LIN {X 0,Y 361.951,Z 263.021,A -85,B 0,C 180,E1 -13113.474,E2 -13113.474} C_VEL
LIN {X 0,Y 361.885,Z 263.028,A -85,B 0,C 180,E1 -13117.143,E2 -13117.143} C_VEL
LIN {X 0,Y 361.906,Z 263.025,A -85,B 0,C 180,E1 -13120.722,E2 -13120.722} C_VEL
LIN {X 0,Y 361.927,Z 263.025,A -85,B 0,C 180,E1 -13123.064,E2 -13123.064} C_VEL
LIN {X 0,Y 361.993,Z 263.017,A -85,B 0,C 180,E1 -13126.526,E2 -13126.526} C_VEL
LIN {X 0,Y 362.025,Z 263.015,A -85,B 0,C 180,E1 -13129.936,E2 -13129.936} C_VEL
LIN {X 0,Y 362.155,Z 262.991,A -85,B 0,C 180,E1 -13133.312,E2 -13133.312} C_VEL
LIN {X 0,Y 362.275,Z 262.98,A -85,B 0,C 180,E1 -13137.775,E2 -13137.775} C_VEL
LIN {X 0,Y 362.421,Z 262.962,A -85,B 0,C 180,E1 -13139.999,E2 -13139.999} C_VEL
LIN {X 0,Y 362.274,Z 262.978,A -85,B 0,C 180,E1 -13142.222,E2 -13142.222} C_VEL
LIN {X 0,Y 362.153,Z 262.994,A -85,B 0,C 180,E1 -13146.685,E2 -13146.685} C_VEL
LIN {X 0,Y 362.021,Z 263.007,A -85,B 0,C 180,E1 -13150.061,E2 -13150.061} C_VEL
LIN {X 0,Y 361.987,Z 263.012,A -85,B 0,C 180,E1 -13153.897,E2 -13153.897} C_VEL
LIN {X 0,Y 361.957,Z 263.018,A -85,B 0,C 180,E1 -13157.938,E2 -13157.938} C_VEL
LIN {X 0,Y 361.891,Z 263.03,A -85,B 0,C 180,E1 -13161.651,E2 -13161.651} C_VEL
LIN {X 0,Y 361.917,Z 263.028,A -85,B 0,C 180,E1 -13165.289,E2 -13165.289} C_VEL
LIN {X 0,Y 361.91,Z 263.028,A -85,B 0,C 180,E1 -13167.777,E2 -13167.777} C_VEL
LIN {X 0,Y 361.834,Z 263.024,A -85,B 0,C 180,E1 -13171.284,E2 -13171.284} C_VEL
LIN {X 0,Y 361.841,Z 263.03,A -85,B 0,C 180,E1 -13174.279,E2 -13174.279} C_VEL
LIN {X 0,Y 361.859,Z 263.037,A -85,B 0,C 180,E1 -13177.224,E2 -13177.224} C_VEL
LIN {X 0,Y 361.892,Z 263.034,A -85,B 0,C 180,E1 -13180.767,E2 -13180.767} C_VEL
LIN {X 0,Y 361.948,Z 263.04,A -85,B 0,C 180,E1 -13184.914,E2 -13184.914} C_VEL
LIN {X 0,Y 364.418,Z 272.898,A -85,B 0,C 180,E1 -13187.831,E2 -13187.831} C_VEL
LIN {X 0,Y 372.996,Z 290.807,A -85,B 0,C 180,E1 -13189.061,E2 -13189.061} C_VEL
LIN {X 0,Y 377.155,Z 300.817,A -85,B 0,C 180,E1 -13189.66,E2 -13189.66} C_VEL
LIN {X 0,Y 377.876,Z 305.295,A -85,B 0,C 180,E1 -13189.822,E2 -13189.822} C_VEL
LIN {X 0,Y 375.211,Z 409.637,A -85,B 0,C 180,E1 -13191.888,E2 -13191.888} C_VEL
LIN {X 0,Y 374.417,Z 423.861,A -85,B 0,C 180,E1 -13192.384,E2 -13192.384} C_VEL
LIN {X 0,Y 373.309,Z 436.994,A -85,B 0,C 180,E1 -13193.041,E2 -13193.041} C_VEL
LIN {X 0,Y 372.043,Z 450.844,A -85,B 0,C 180,E1 -13193.989,E2 -13193.989} C_VEL
LIN {X 0,Y 370.563,Z 463.295,A -85,B 0,C 180,E1 -13195.075,E2 -13195.075} C_VEL
LIN {X 0,Y 369.18,Z 473.466,A -85,B 0,C 180,E1 -13196.165,E2 -13196.165} C_VEL
LIN {X 0,Y 367.475,Z 484.71,A -85,B 0,C 180,E1 -13197.623,E2 -13197.623} C_VEL
LIN {X 0,Y 366.018,Z 494.031,A -85,B 0,C 180,E1 -13199.095,E2 -13199.095} C_VEL
LIN {X 0,Y 364.568,Z 503.314,A -85,B 0,C 180,E1 -13200.873,E2 -13200.873} C_VEL
LIN {X 0,Y 363.209,Z 511.817,A -85,B 0,C 180,E1 -13202.88,E2 -13202.88} C_VEL
LIN {X 0,Y 362.229,Z 518.114,A -85,B 0,C 180,E1 -13204.733,E2 -13204.733} C_VEL
LIN {X 0,Y 361.511,Z 523.028,A -85,B 0,C 180,E1 -13206.533,E2 -13206.533} C_VEL
LIN {X 0,Y 360.993,Z 526.84,A -85,B 0,C 180,E1 -13208.291,E2 -13208.291} C_VEL
LIN {X 0,Y 360.753,Z 528.882,A -85,B 0,C 180,E1 -13209.473,E2 -13209.473} C_VEL
LIN {X 0,Y 360.334,Z 531.796,A -85,B 0,C 180,E1 -13211.817,E2 -13211.817} C_VEL
LIN {X 0,Y 360.169,Z 533.243,A -85,B 0,C 180,E1 -13214.147,E2 -13214.147} C_VEL
LIN {X 0,Y 360.14,Z 533.273,A -85,B 0,C 180,E1 -13216.457,E2 -13216.457} C_VEL
LIN {X 0,Y 360.223,Z 532.756,A -85,B 0,C 180,E1 -13217.608,E2 -13217.608} C_VEL
LIN {X 0,Y 360.232,Z 530.689,A -85,B 0,C 180,E1 -13219.888,E2 -13219.888} C_VEL
LIN {X 0,Y 360.554,Z 527.2,A -85,B 0,C 180,E1 -13222.158,E2 -13222.158} C_VEL
LIN {X 0,Y 360.956,Z 522.221,A -85,B 0,C 180,E1 -13224.414,E2 -13224.414} C_VEL
LIN {X 0,Y 361.337,Z 517.421,A -85,B 0,C 180,E1 -13226.097,E2 -13226.097} C_VEL
LIN {X 0,Y 361.974,Z 510.498,A -85,B 0,C 180,E1 -13228.053,E2 -13228.053} C_VEL
LIN {X 0,Y 362.819,Z 503.263,A -85,B 0,C 180,E1 -13229.723,E2 -13229.723} C_VEL
LIN {X 0,Y 363.876,Z 494.569,A -85,B 0,C 180,E1 -13231.384,E2 -13231.384} C_VEL
LIN {X 0,Y 365.098,Z 484.058,A -85,B 0,C 180,E1 -13233.035,E2 -13233.035} C_VEL
LIN {X 0,Y 366.459,Z 472.289,A -85,B 0,C 180,E1 -13234.537,E2 -13234.537} C_VEL
LIN {X 0,Y 367.69,Z 460.24,A -85,B 0,C 180,E1 -13235.784,E2 -13235.784} C_VEL
LIN {X 0,Y 368.854,Z 447.486,A -85,B 0,C 180,E1 -13236.839,E2 -13236.839} C_VEL
LIN {X 0,Y 369.768,Z 433.835,A -85,B 0,C 180,E1 -13237.714,E2 -13237.714} C_VEL
LIN {X 0,Y 370.561,Z 419.368,A -85,B 0,C 180,E1 -13238.384,E2 -13238.384} C_VEL
LIN {X 0,Y 371.08,Z 405.045,A -85,B 0,C 180,E1 -13238.818,E2 -13238.818} C_VEL
LIN {X 0,Y 371.751,Z 371.974,A -85,B 0,C 180,E1 -13239.465,E2 -13239.465} C_VEL
LIN {X 0,Y 371.242,Z 366.164,A -85,B 0,C 180,E1 -13239.612,E2 -13239.612} C_VEL
LIN {X 0,Y 366.276,Z 347.449,A -85,B 0,C 180,E1 -13240.285,E2 -13240.285} C_VEL
LIN {X 0,Y 365.76,Z 341.639,A -85,B 0,C 180,E1 -13240.437,E2 -13240.437} C_VEL
LIN {X 0,Y 366.376,Z 302.629,A -85,B 0,C 180,E1 -13241.213,E2 -13241.213} C_VEL
LIN {X 0,Y 363.787,Z 291.177,A -85,B 0,C 180,E1 -13241.617,E2 -13241.617} C_VEL
LIN {X 0,Y 356.731,Z 272.196,A -85,B 0,C 180,E1 -13242.516,E2 -13242.516} C_VEL
LIN {X 0,Y 354.914,Z 263.908,A -85,B 0,C 180,E1 -13244.744,E2 -13244.744} C_VEL
LIN {X 0,Y 354.895,Z 263.9,A -85,B 0,C 180,E1 -13248.472,E2 -13248.472} C_VEL
LIN {X 0,Y 354.826,Z 263.911,A -85,B 0,C 180,E1 -13252.106,E2 -13252.106} C_VEL
LIN {X 0,Y 354.886,Z 263.905,A -85,B 0,C 180,E1 -13255.828,E2 -13255.828} C_VEL
LIN {X 0,Y 354.842,Z 263.911,A -85,B 0,C 180,E1 -13259.679,E2 -13259.679} C_VEL
LIN {X 0,Y 354.793,Z 263.916,A -85,B 0,C 180,E1 -13263.703,E2 -13263.703} C_VEL
LIN {X 0,Y 354.789,Z 263.912,A -85,B 0,C 180,E1 -13266.46,E2 -13266.46} C_VEL
LIN {X 0,Y 354.812,Z 263.916,A -85,B 0,C 180,E1 -13269.424,E2 -13269.424} C_VEL
LIN {X 0,Y 354.83,Z 263.909,A -85,B 0,C 180,E1 -13272.877,E2 -13272.877} C_VEL
LIN {X 0,Y 354.853,Z 263.904,A -85,B 0,C 180,E1 -13276.12,E2 -13276.12} C_VEL
LIN {X 0,Y 354.844,Z 263.911,A -85,B 0,C 180,E1 -13279.19,E2 -13279.19} C_VEL
LIN {X 0,Y 354.797,Z 263.912,A -85,B 0,C 180,E1 -13282.403,E2 -13282.403} C_VEL
LIN {X 0,Y 354.801,Z 263.914,A -85,B 0,C 180,E1 -13284.942,E2 -13284.942} C_VEL
LIN {X 0,Y 354.782,Z 263.914,A -85,B 0,C 180,E1 -13288.406,E2 -13288.406} C_VEL
LIN {X 0,Y 354.843,Z 263.906,A -85,B 0,C 180,E1 -13291.621,E2 -13291.621} C_VEL
LIN {X 0,Y 354.889,Z 263.9,A -85,B 0,C 180,E1 -13294.174,E2 -13294.174} C_VEL
LIN {X 0,Y 354.824,Z 263.908,A -85,B 0,C 180,E1 -13297.895,E2 -13297.895} C_VEL
LIN {X 0,Y 354.913,Z 263.897,A -85,B 0,C 180,E1 -13301.893,E2 -13301.893} C_VEL
LIN {X 0,Y 354.934,Z 263.895,A -85,B 0,C 180,E1 -13305.983,E2 -13305.983} C_VEL
LIN {X 0,Y 354.97,Z 263.89,A -85,B 0,C 180,E1 -13309.737,E2 -13309.737} C_VEL
LIN {X 0,Y 355.119,Z 263.872,A -85,B 0,C 180,E1 -13313.182,E2 -13313.182} C_VEL
LIN {X 0,Y 355.239,Z 263.857,A -85,B 0,C 180,E1 -13317.734,E2 -13317.734} C_VEL
LIN {X 0,Y 355.39,Z 263.839,A -85,B 0,C 180,E1 -13320.002,E2 -13320.002} C_VEL
LIN {X 0,Y 355.239,Z 263.86,A -85,B 0,C 180,E1 -13322.269,E2 -13322.269} C_VEL
LIN {X 0,Y 355.12,Z 263.873,A -85,B 0,C 180,E1 -13326.821,E2 -13326.821} C_VEL
LIN {X 0,Y 354.973,Z 263.896,A -85,B 0,C 180,E1 -13330.266,E2 -13330.266} C_VEL
LIN {X 0,Y 354.939,Z 263.897,A -85,B 0,C 180,E1 -13334.02,E2 -13334.02} C_VEL
LIN {X 0,Y 354.919,Z 263.902,A -85,B 0,C 180,E1 -13338.11,E2 -13338.11} C_VEL
LIN {X 0,Y 354.814,Z 263.915,A -85,B 0,C 180,E1 -13342.109,E2 -13342.109} C_VEL
LIN {X 0,Y 354.896,Z 263.903,A -85,B 0,C 180,E1 -13345.829,E2 -13345.829} C_VEL
LIN {X 0,Y 354.853,Z 263.908,A -85,B 0,C 180,E1 -13349.68,E2 -13349.68} C_VEL
LIN {X 0,Y 354.83,Z 263.912,A -85,B 0,C 180,E1 -13353.684,E2 -13353.684} C_VEL
LIN {X 0,Y 354.798,Z 263.912,A -85,B 0,C 180,E1 -13356.461,E2 -13356.461} C_VEL
LIN {X 0,Y 354.824,Z 263.911,A -85,B 0,C 180,E1 -13359.425,E2 -13359.425} C_VEL
LIN {X 0,Y 354.788,Z 263.913,A -85,B 0,C 180,E1 -13362.868,E2 -13362.868} C_VEL
LIN {X 0,Y 354.768,Z 263.917,A -85,B 0,C 180,E1 -13366.105,E2 -13366.105} C_VEL
LIN {X 0,Y 354.788,Z 263.915,A -85,B 0,C 180,E1 -13369.18,E2 -13369.18} C_VEL
LIN {X 0,Y 354.808,Z 263.91,A -85,B 0,C 180,E1 -13372.404,E2 -13372.404} C_VEL
LIN {X 0,Y 354.814,Z 263.911,A -85,B 0,C 180,E1 -13374.942,E2 -13374.942} C_VEL
LIN {X 0,Y 354.846,Z 264.002,A -85,B 0,C 180,E1 -13377.589,E2 -13377.589} C_VEL
LIN {X 0,Y 357.921,Z 277.781,A -85,B 0,C 180,E1 -13380.924,E2 -13380.924} C_VEL
LIN {X 0,Y 359.764,Z 286.653,A -85,B 0,C 180,E1 -13382.988,E2 -13382.988} C_VEL
LIN {X 0,Y 359.785,Z 290.384,A -85,B 0,C 180,E1 -13383.74,E2 -13383.74} C_VEL
LIN {X 0,Y 366.128,Z 328.545,A -85,B 0,C 180,E1 -13384.945,E2 -13384.945} C_VEL
LIN {X 0,Y 364.125,Z 427.883,A -85,B 0,C 180,E1 -13386.918,E2 -13386.918} C_VEL
LIN {X 0,Y 363.381,Z 442.676,A -85,B 0,C 180,E1 -13387.432,E2 -13387.432} C_VEL
LIN {X 0,Y 362.317,Z 456.75,A -85,B 0,C 180,E1 -13388.15,E2 -13388.15} C_VEL
LIN {X 0,Y 361.201,Z 470.732,A -85,B 0,C 180,E1 -13389.125,E2 -13389.125} C_VEL
LIN {X 0,Y 359.782,Z 483.977,A -85,B 0,C 180,E1 -13390.308,E2 -13390.308} C_VEL
LIN {X 0,Y 358.365,Z 496.401,A -85,B 0,C 180,E1 -13391.713,E2 -13391.713} C_VEL
LIN {X 0,Y 357.116,Z 506.619,A -85,B 0,C 180,E1 -13393.126,E2 -13393.126} C_VEL
LIN {X 0,Y 355.983,Z 516.769,A -85,B 0,C 180,E1 -13394.836,E2 -13394.836} C_VEL
LIN {X 0,Y 355.17,Z 525.186,A -85,B 0,C 180,E1 -13396.556,E2 -13396.556} C_VEL
LIN {X 0,Y 354.276,Z 533.205,A -85,B 0,C 180,E1 -13398.558,E2 -13398.558} C_VEL
LIN {X 0,Y 353.783,Z 538.828,A -85,B 0,C 180,E1 -13400.279,E2 -13400.279} C_VEL
LIN {X 0,Y 353.417,Z 544.71,A -85,B 0,C 180,E1 -13402.573,E2 -13402.573} C_VEL
LIN {X 0,Y 353.265,Z 548.085,A -85,B 0,C 180,E1 -13404.291,E2 -13404.291} C_VEL
LIN {X 0,Y 353.207,Z 551.233,A -85,B 0,C 180,E1 -13406.578,E2 -13406.578} C_VEL
LIN {X 0,Y 353.221,Z 552.988,A -85,B 0,C 180,E1 -13408.86,E2 -13408.86} C_VEL
LIN {X 0,Y 353.263,Z 553.359,A -85,B 0,C 180,E1 -13410,E2 -13410} C_VEL
LIN {X 0,Y 353.167,Z 553.092,A -85,B 0,C 180,E1 -13412.281,E2 -13412.281} C_VEL
LIN {X 0,Y 353.242,Z 551.497,A -85,B 0,C 180,E1 -13414.564,E2 -13414.564} C_VEL
LIN {X 0,Y 353.396,Z 548.542,A -85,B 0,C 180,E1 -13416.853,E2 -13416.853} C_VEL
LIN {X 0,Y 353.775,Z 544.152,A -85,B 0,C 180,E1 -13419.144,E2 -13419.144} C_VEL
LIN {X 0,Y 354.421,Z 538.215,A -85,B 0,C 180,E1 -13421.437,E2 -13421.437} C_VEL
LIN {X 0,Y 355.514,Z 531.558,A -85,B 0,C 180,E1 -13423.431,E2 -13423.431} C_VEL
LIN {X 0,Y 356.675,Z 523.31,A -85,B 0,C 180,E1 -13425.426,E2 -13425.426} C_VEL
LIN {X 0,Y 358.084,Z 514.738,A -85,B 0,C 180,E1 -13427.121,E2 -13427.121} C_VEL
LIN {X 0,Y 359.812,Z 504.379,A -85,B 0,C 180,E1 -13428.801,E2 -13428.801} C_VEL
LIN {X 0,Y 361.661,Z 492.828,A -85,B 0,C 180,E1 -13430.325,E2 -13430.325} C_VEL
LIN {X 0,Y 363.336,Z 481.321,A -85,B 0,C 180,E1 -13431.562,E2 -13431.562} C_VEL
LIN {X 0,Y 364.933,Z 468.715,A -85,B 0,C 180,E1 -13432.653,E2 -13432.653} C_VEL
LIN {X 0,Y 366.396,Z 455.701,A -85,B 0,C 180,E1 -13433.528,E2 -13433.528} C_VEL
LIN {X 0,Y 367.728,Z 441.697,A -85,B 0,C 180,E1 -13434.224,E2 -13434.224} C_VEL
LIN {X 0,Y 368.599,Z 428.135,A -85,B 0,C 180,E1 -13434.688,E2 -13434.688} C_VEL
LIN {X 0,Y 371.103,Z 329.531,A -85,B 0,C 180,E1 -13436.683,E2 -13436.683} C_VEL
LIN {X 0,Y 366.385,Z 305.41,A -85,B 0,C 180,E1 -13437.663,E2 -13437.663} C_VEL
LIN {X 0,Y 364.205,Z 296.489,A -85,B 0,C 180,E1 -13438.077,E2 -13438.077} C_VEL
LIN {X 0,Y 361.196,Z 289.435,A -85,B 0,C 180,E1 -13438.551,E2 -13438.551} C_VEL
LIN {X 0,Y 358.485,Z 277.757,A -85,B 0,C 180,E1 -13441.628,E2 -13441.628} C_VEL
LIN {X 0,Y 355.393,Z 265.851,A -85,B 0,C 180,E1 -13444.992,E2 -13444.992} C_VEL
LIN {X 0,Y 354.837,Z 263.916,A -85,B 0,C 180,E1 -13445.601,E2 -13445.601} C_VEL
LIN {X 0,Y 354.825,Z 263.917,A -85,B 0,C 180,E1 -13449.422,E2 -13449.422} C_VEL
LIN {X 0,Y 354.834,Z 263.912,A -85,B 0,C 180,E1 -13452.874,E2 -13452.874} C_VEL
LIN {X 0,Y 354.783,Z 263.916,A -85,B 0,C 180,E1 -13456.105,E2 -13456.105} C_VEL
LIN {X 0,Y 354.786,Z 263.916,A -85,B 0,C 180,E1 -13459.177,E2 -13459.177} C_VEL
LIN {X 0,Y 354.805,Z 263.909,A -85,B 0,C 180,E1 -13462.401,E2 -13462.401} C_VEL
LIN {X 0,Y 354.809,Z 263.893,A -85,B 0,C 180,E1 -13464.939,E2 -13464.939} C_VEL
LIN {X 0,Y 354.79,Z 263.909,A -85,B 0,C 180,E1 -13468.404,E2 -13468.404} C_VEL
LIN {X 0,Y 354.85,Z 263.906,A -85,B 0,C 180,E1 -13471.618,E2 -13471.618} C_VEL
LIN {X 0,Y 354.895,Z 263.903,A -85,B 0,C 180,E1 -13474.171,E2 -13474.171} C_VEL
LIN {X 0,Y 354.83,Z 263.913,A -85,B 0,C 180,E1 -13477.892,E2 -13477.892} C_VEL
LIN {X 0,Y 354.918,Z 263.901,A -85,B 0,C 180,E1 -13481.89,E2 -13481.89} C_VEL
LIN {X 0,Y 354.937,Z 263.898,A -85,B 0,C 180,E1 -13485.98,E2 -13485.98} C_VEL
LIN {X 0,Y 354.971,Z 263.894,A -85,B 0,C 180,E1 -13489.734,E2 -13489.734} C_VEL
LIN {X 0,Y 355.119,Z 263.866,A -85,B 0,C 180,E1 -13493.179,E2 -13493.179} C_VEL
LIN {X 0,Y 355.238,Z 263.855,A -85,B 0,C 180,E1 -13497.731,E2 -13497.731} C_VEL
LIN {X 0,Y 355.391,Z 263.838,A -85,B 0,C 180,E1 -13499.998,E2 -13499.998} C_VEL
LIN {X 0,Y 355.237,Z 263.855,A -85,B 0,C 180,E1 -13502.266,E2 -13502.266} C_VEL
LIN {X 0,Y 355.117,Z 263.871,A -85,B 0,C 180,E1 -13506.818,E2 -13506.818} C_VEL
LIN {X 0,Y 354.968,Z 263.886,A -85,B 0,C 180,E1 -13510.263,E2 -13510.263} C_VEL
LIN {X 0,Y 354.932,Z 263.891,A -85,B 0,C 180,E1 -13514.017,E2 -13514.017} C_VEL
LIN {X 0,Y 354.913,Z 263.896,A -85,B 0,C 180,E1 -13518.108,E2 -13518.108} C_VEL
LIN {X 0,Y 354.833,Z 263.909,A -85,B 0,C 180,E1 -13522.104,E2 -13522.104} C_VEL
LIN {X 0,Y 354.888,Z 263.903,A -85,B 0,C 180,E1 -13525.826,E2 -13525.826} C_VEL
LIN {X 0,Y 354.842,Z 263.901,A -85,B 0,C 180,E1 -13529.677,E2 -13529.677} C_VEL
LIN {X 0,Y 354.793,Z 263.915,A -85,B 0,C 180,E1 -13533.701,E2 -13533.701} C_VEL
LIN {X 0,Y 354.788,Z 263.912,A -85,B 0,C 180,E1 -13536.458,E2 -13536.458} C_VEL
LIN {X 0,Y 354.811,Z 263.905,A -85,B 0,C 180,E1 -13539.423,E2 -13539.423} C_VEL
LIN {X 0,Y 354.828,Z 263.907,A -85,B 0,C 180,E1 -13542.876,E2 -13542.876} C_VEL
LIN {X 0,Y 354.919,Z 264.059,A -85,B 0,C 180,E1 -13544.327,E2 -13544.327} C_VEL
LIN {X 0,Y 357.304,Z 273.246,A -85,B 0,C 180,E1 -13547.109,E2 -13547.109} C_VEL
LIN {X 0,Y 366.119,Z 291.157,A -85,B 0,C 180,E1 -13548.418,E2 -13548.418} C_VEL
LIN {X 0,Y 371.246,Z 303.218,A -85,B 0,C 180,E1 -13549.176,E2 -13549.176} C_VEL
LIN {X 0,Y 371.747,Z 306.001,A -85,B 0,C 180,E1 -13549.284,E2 -13549.284} C_VEL
LIN {X 0,Y 368.982,Z 409.593,A -85,B 0,C 180,E1 -13551.367,E2 -13551.367} C_VEL
LIN {X 0,Y 368.105,Z 424.319,A -85,B 0,C 180,E1 -13551.888,E2 -13551.888} C_VEL
LIN {X 0,Y 366.87,Z 438.537,A -85,B 0,C 180,E1 -13552.626,E2 -13552.626} C_VEL
LIN {X 0,Y 365.619,Z 451.321,A -85,B 0,C 180,E1 -13553.528,E2 -13553.528} C_VEL
LIN {X 0,Y 364.088,Z 463.555,A -85,B 0,C 180,E1 -13554.614,E2 -13554.614} C_VEL
LIN {X 0,Y 362.552,Z 474.341,A -85,B 0,C 180,E1 -13555.796,E2 -13555.796} C_VEL
LIN {X 0,Y 360.778,Z 485.47,A -85,B 0,C 180,E1 -13557.278,E2 -13557.278} C_VEL
LIN {X 0,Y 359.246,Z 494.693,A -85,B 0,C 180,E1 -13558.774,E2 -13558.774} C_VEL
LIN {X 0,Y 357.716,Z 503.898,A -85,B 0,C 180,E1 -13560.583,E2 -13560.583} C_VEL
LIN {X 0,Y 356.333,Z 512.078,A -85,B 0,C 180,E1 -13562.561,E2 -13562.561} C_VEL
LIN {X 0,Y 355.403,Z 517.622,A -85,B 0,C 180,E1 -13564.213,E2 -13564.213} C_VEL
LIN {X 0,Y 354.57,Z 522.958,A -85,B 0,C 180,E1 -13566.16,E2 -13566.16} C_VEL
LIN {X 0,Y 353.878,Z 527.737,A -85,B 0,C 180,E1 -13568.445,E2 -13568.445} C_VEL
LIN {X 0,Y 353.491,Z 530.451,A -85,B 0,C 180,E1 -13570.246,E2 -13570.246} C_VEL
LIN {X 0,Y 353.179,Z 532.748,A -85,B 0,C 180,E1 -13572.634,E2 -13572.634} C_VEL
LIN {X 0,Y 353.04,Z 533.608,A -85,B 0,C 180,E1 -13575.002,E2 -13575.002} C_VEL
LIN {X 0,Y 353.124,Z 533.069,A -85,B 0,C 180,E1 -13577.354,E2 -13577.354} C_VEL
LIN {X 0,Y 353.129,Z 531.156,A -85,B 0,C 180,E1 -13579.682,E2 -13579.682} C_VEL
LIN {X 0,Y 353.44,Z 527.799,A -85,B 0,C 180,E1 -13581.999,E2 -13581.999} C_VEL
LIN {X 0,Y 353.675,Z 524.86,A -85,B 0,C 180,E1 -13583.478,E2 -13583.478} C_VEL
LIN {X 0,Y 354.03,Z 519.936,A -85,B 0,C 180,E1 -13585.446,E2 -13585.446} C_VEL
LIN {X 0,Y 354.657,Z 513.585,A -85,B 0,C 180,E1 -13587.445,E2 -13587.445} C_VEL
LIN {X 0,Y 355.611,Z 505.686,A -85,B 0,C 180,E1 -13589.434,E2 -13589.434} C_VEL
LIN {X 0,Y 356.592,Z 497.444,A -85,B 0,C 180,E1 -13591.129,E2 -13591.129} C_VEL
LIN {X 0,Y 357.806,Z 487.525,A -85,B 0,C 180,E1 -13592.815,E2 -13592.815} C_VEL
LIN {X 0,Y 359.162,Z 476.493,A -85,B 0,C 180,E1 -13594.349,E2 -13594.349} C_VEL
LIN {X 0,Y 360.387,Z 465.534,A -85,B 0,C 180,E1 -13595.596,E2 -13595.596} C_VEL
LIN {X 0,Y 361.491,Z 453.705,A -85,B 0,C 180,E1 -13596.699,E2 -13596.699} C_VEL
LIN {X 0,Y 362.593,Z 440.692,A -85,B 0,C 180,E1 -13597.658,E2 -13597.658} C_VEL
LIN {X 0,Y 363.51,Z 426.527,A -85,B 0,C 180,E1 -13598.442,E2 -13598.442} C_VEL
LIN {X 0,Y 364.127,Z 412.525,A -85,B 0,C 180,E1 -13598.987,E2 -13598.987} C_VEL
LIN {X 0,Y 364.629,Z 393.271,A -85,B 0,C 180,E1 -13599.429,E2 -13599.429} C_VEL
LIN {X 0,Y 365.76,Z 341.639,A -85,B 0,C 180,E1 -13600.437,E2 -13600.437} C_VEL
LIN {X 0,Y 365.258,Z 335.834,A -85,B 0,C 180,E1 -13600.588,E2 -13600.588} C_VEL
LIN {X 0,Y 360.352,Z 317.13,A -85,B 0,C 180,E1 -13601.285,E2 -13601.285} C_VEL
LIN {X 0,Y 359.783,Z 311.326,A -85,B 0,C 180,E1 -13601.444,E2 -13601.444} C_VEL
LIN {X 0,Y 359.816,Z 303.66,A -85,B 0,C 180,E1 -13601.605,E2 -13601.605} C_VEL
LIN {X 0,Y 357.411,Z 293.434,A -85,B 0,C 180,E1 -13601.98,E2 -13601.98} C_VEL
LIN {X 0,Y 349.57,Z 272.415,A -85,B 0,C 180,E1 -13602.998,E2 -13602.998} C_VEL
LIN {X 0,Y 347.864,Z 264.783,A -85,B 0,C 180,E1 -13605.098,E2 -13605.098} C_VEL
LIN {X 0,Y 347.846,Z 264.778,A -85,B 0,C 180,E1 -13608.86,E2 -13608.86} C_VEL
LIN {X 0,Y 347.764,Z 264.788,A -85,B 0,C 180,E1 -13612.58,E2 -13612.58} C_VEL
LIN {X 0,Y 347.799,Z 264.785,A -85,B 0,C 180,E1 -13615.109,E2 -13615.109} C_VEL
LIN {X 0,Y 347.8,Z 264.789,A -85,B 0,C 180,E1 -13617.694,E2 -13617.694} C_VEL
LIN {X 0,Y 347.752,Z 264.789,A -85,B 0,C 180,E1 -13620.347,E2 -13620.347} C_VEL
LIN {X 0,Y 347.731,Z 264.792,A -85,B 0,C 180,E1 -13624.465,E2 -13624.465} C_VEL
LIN {X 0,Y 347.766,Z 264.789,A -85,B 0,C 180,E1 -13627.991,E2 -13627.991} C_VEL
LIN {X 0,Y 347.772,Z 264.788,A -85,B 0,C 180,E1 -13631.826,E2 -13631.826} C_VEL
LIN {X 0,Y 347.818,Z 264.784,A -85,B 0,C 180,E1 -13635.007,E2 -13635.007} C_VEL
LIN {X 0,Y 347.773,Z 264.786,A -85,B 0,C 180,E1 -13638.392,E2 -13638.392} C_VEL
LIN {X 0,Y 347.765,Z 264.787,A -85,B 0,C 180,E1 -13642.012,E2 -13642.012} C_VEL
LIN {X 0,Y 347.733,Z 264.793,A -85,B 0,C 180,E1 -13645.537,E2 -13645.537} C_VEL
LIN {X 0,Y 347.754,Z 264.79,A -85,B 0,C 180,E1 -13649.655,E2 -13649.655} C_VEL
LIN {X 0,Y 347.842,Z 264.78,A -85,B 0,C 180,E1 -13652.746,E2 -13652.746} C_VEL
LIN {X 0,Y 347.778,Z 264.786,A -85,B 0,C 180,E1 -13656.163,E2 -13656.163} C_VEL
LIN {X 0,Y 347.803,Z 264.783,A -85,B 0,C 180,E1 -13659.911,E2 -13659.911} C_VEL
LIN {X 0,Y 347.857,Z 264.778,A -85,B 0,C 180,E1 -13662.361,E2 -13662.361} C_VEL
LIN {X 0,Y 347.889,Z 264.772,A -85,B 0,C 180,E1 -13665.972,E2 -13665.972} C_VEL
LIN {X 0,Y 347.92,Z 264.768,A -85,B 0,C 180,E1 -13669.527,E2 -13669.527} C_VEL
LIN {X 0,Y 348.085,Z 264.748,A -85,B 0,C 180,E1 -13673.044,E2 -13673.044} C_VEL
LIN {X 0,Y 348.201,Z 264.733,A -85,B 0,C 180,E1 -13677.688,E2 -13677.688} C_VEL
LIN {X 0,Y 348.339,Z 264.717,A -85,B 0,C 180,E1 -13680.002,E2 -13680.002} C_VEL
LIN {X 0,Y 348.202,Z 264.737,A -85,B 0,C 180,E1 -13682.315,E2 -13682.315} C_VEL
LIN {X 0,Y 348.086,Z 264.749,A -85,B 0,C 180,E1 -13686.96,E2 -13686.96} C_VEL
LIN {X 0,Y 347.923,Z 264.771,A -85,B 0,C 180,E1 -13690.476,E2 -13690.476} C_VEL
LIN {X 0,Y 347.895,Z 264.775,A -85,B 0,C 180,E1 -13694.151,E2 -13694.151} C_VEL
LIN {X 0,Y 347.888,Z 264.777,A -85,B 0,C 180,E1 -13698.292,E2 -13698.292} C_VEL
LIN {X 0,Y 347.765,Z 264.789,A -85,B 0,C 180,E1 -13701.628,E2 -13701.628} C_VEL
LIN {X 0,Y 347.809,Z 264.782,A -85,B 0,C 180,E1 -13705.11,E2 -13705.11} C_VEL
LIN {X 0,Y 347.81,Z 264.785,A -85,B 0,C 180,E1 -13707.695,E2 -13707.695} C_VEL
LIN {X 0,Y 347.769,Z 264.789,A -85,B 0,C 180,E1 -13710.347,E2 -13710.347} C_VEL
LIN {X 0,Y 347.747,Z 264.794,A -85,B 0,C 180,E1 -13714.045,E2 -13714.045} C_VEL
LIN {X 0,Y 347.762,Z 264.79,A -85,B 0,C 180,E1 -13717.322,E2 -13717.322} C_VEL
LIN {X 0,Y 347.732,Z 264.793,A -85,B 0,C 180,E1 -13720.298,E2 -13720.298} C_VEL
LIN {X 0,Y 347.724,Z 264.796,A -85,B 0,C 180,E1 -13723.409,E2 -13723.409} C_VEL
LIN {X 0,Y 347.726,Z 264.793,A -85,B 0,C 180,E1 -13726.688,E2 -13726.688} C_VEL
LIN {X 0,Y 347.749,Z 264.791,A -85,B 0,C 180,E1 -13730.174,E2 -13730.174} C_VEL
LIN {X 0,Y 347.763,Z 264.788,A -85,B 0,C 180,E1 -13732.68,E2 -13732.68} C_VEL
LIN {X 0,Y 347.751,Z 264.797,A -85,B 0,C 180,E1 -13735.957,E2 -13735.957} C_VEL
LIN {X 0,Y 347.799,Z 264.909,A -85,B 0,C 180,E1 -13737.217,E2 -13737.217} C_VEL
LIN {X 0,Y 350.903,Z 278.597,A -85,B 0,C 180,E1 -13740.614,E2 -13740.614} C_VEL
LIN {X 0,Y 352.919,Z 288.861,A -85,B 0,C 180,E1 -13743.046,E2 -13743.046} C_VEL
LIN {X 0,Y 352.97,Z 289.824,A -85,B 0,C 180,E1 -13743.262,E2 -13743.262} C_VEL
LIN {X 0,Y 359.484,Z 330.124,A -85,B 0,C 180,E1 -13744.568,E2 -13744.568} C_VEL
LIN {X 0,Y 357.446,Z 427.588,A -85,B 0,C 180,E1 -13746.538,E2 -13746.538} C_VEL
LIN {X 0,Y 356.678,Z 442.42,A -85,B 0,C 180,E1 -13747.06,E2 -13747.06} C_VEL
LIN {X 0,Y 355.588,Z 456.509,A -85,B 0,C 180,E1 -13747.791,E2 -13747.791} C_VEL
LIN {X 0,Y 354.384,Z 470.303,A -85,B 0,C 180,E1 -13748.764,E2 -13748.764} C_VEL
LIN {X 0,Y 352.989,Z 483.022,A -85,B 0,C 180,E1 -13749.913,E2 -13749.913} C_VEL
LIN {X 0,Y 351.679,Z 494.468,A -85,B 0,C 180,E1 -13751.202,E2 -13751.202} C_VEL
LIN {X 0,Y 350.524,Z 503.993,A -85,B 0,C 180,E1 -13752.498,E2 -13752.498} C_VEL
LIN {X 0,Y 349.197,Z 514.61,A -85,B 0,C 180,E1 -13754.235,E2 -13754.235} C_VEL
LIN {X 0,Y 348.311,Z 523.371,A -85,B 0,C 180,E1 -13755.988,E2 -13755.988} C_VEL
LIN {X 0,Y 347.364,Z 531.728,A -85,B 0,C 180,E1 -13758.031,E2 -13758.031} C_VEL
LIN {X 0,Y 346.72,Z 538.427,A -85,B 0,C 180,E1 -13760.079,E2 -13760.079} C_VEL
LIN {X 0,Y 346.347,Z 544.36,A -85,B 0,C 180,E1 -13762.421,E2 -13762.421} C_VEL
LIN {X 0,Y 346.185,Z 547.775,A -85,B 0,C 180,E1 -13764.174,E2 -13764.174} C_VEL
LIN {X 0,Y 346.13,Z 550.967,A -85,B 0,C 180,E1 -13766.508,E2 -13766.508} C_VEL
LIN {X 0,Y 346.122,Z 552.759,A -85,B 0,C 180,E1 -13768.836,E2 -13768.836} C_VEL
LIN {X 0,Y 346.165,Z 553.149,A -85,B 0,C 180,E1 -13770,E2 -13770} C_VEL
LIN {X 0,Y 346.078,Z 552.921,A -85,B 0,C 180,E1 -13772.328,E2 -13772.328} C_VEL
LIN {X 0,Y 346.143,Z 551.365,A -85,B 0,C 180,E1 -13774.658,E2 -13774.658} C_VEL
LIN {X 0,Y 346.322,Z 548.452,A -85,B 0,C 180,E1 -13776.993,E2 -13776.993} C_VEL
LIN {X 0,Y 346.721,Z 544.109,A -85,B 0,C 180,E1 -13779.332,E2 -13779.332} C_VEL
LIN {X 0,Y 347.437,Z 538.219,A -85,B 0,C 180,E1 -13781.67,E2 -13781.67} C_VEL
LIN {X 0,Y 348.558,Z 531.616,A -85,B 0,C 180,E1 -13783.704,E2 -13783.704} C_VEL
LIN {X 0,Y 349.815,Z 523.451,A -85,B 0,C 180,E1 -13785.737,E2 -13785.737} C_VEL
LIN {X 0,Y 351.281,Z 514.944,A -85,B 0,C 180,E1 -13787.463,E2 -13787.463} C_VEL
LIN {X 0,Y 353.112,Z 504.674,A -85,B 0,C 180,E1 -13789.171,E2 -13789.171} C_VEL
LIN {X 0,Y 355.03,Z 493.236,A -85,B 0,C 180,E1 -13790.722,E2 -13790.722} C_VEL
LIN {X 0,Y 356.918,Z 480.614,A -85,B 0,C 180,E1 -13792.106,E2 -13792.106} C_VEL
LIN {X 0,Y 358.676,Z 467.71,A -85,B 0,C 180,E1 -13793.224,E2 -13793.224} C_VEL
LIN {X 0,Y 360.198,Z 454.489,A -85,B 0,C 180,E1 -13794.111,E2 -13794.111} C_VEL
LIN {X 0,Y 361.474,Z 440.904,A -85,B 0,C 180,E1 -13794.785,E2 -13794.785} C_VEL
LIN {X 0,Y 362.426,Z 426.989,A -85,B 0,C 180,E1 -13795.252,E2 -13795.252} C_VEL
LIN {X 0,Y 364.966,Z 330.613,A -85,B 0,C 180,E1 -13797.225,E2 -13797.225} C_VEL
LIN {X 0,Y 360.245,Z 306.351,A -85,B 0,C 180,E1 -13798.241,E2 -13798.241} C_VEL
LIN {X 0,Y 358.522,Z 299.42,A -85,B 0,C 180,E1 -13798.577,E2 -13798.577} C_VEL
LIN {X 0,Y 353.912,Z 289.071,A -85,B 0,C 180,E1 -13799.338,E2 -13799.338} C_VEL
LIN {X 0,Y 351.633,Z 279.343,A -85,B 0,C 180,E1 -13801.981,E2 -13801.981} C_VEL
LIN {X 0,Y 348.561,Z 267.736,A -85,B 0,C 180,E1 -13805.36,E2 -13805.36} C_VEL
LIN {X 0,Y 347.779,Z 264.797,A -85,B 0,C 180,E1 -13806.298,E2 -13806.298} C_VEL
LIN {X 0,Y 347.794,Z 264.781,A -85,B 0,C 180,E1 -13810.287,E2 -13810.287} C_VEL
LIN {X 0,Y 347.783,Z 264.788,A -85,B 0,C 180,E1 -13813.397,E2 -13813.397} C_VEL
LIN {X 0,Y 347.728,Z 264.796,A -85,B 0,C 180,E1 -13816.684,E2 -13816.684} C_VEL
LIN {X 0,Y 347.746,Z 264.791,A -85,B 0,C 180,E1 -13820.172,E2 -13820.172} C_VEL
LIN {X 0,Y 347.759,Z 264.784,A -85,B 0,C 180,E1 -13822.678,E2 -13822.678} C_VEL
LIN {X 0,Y 347.746,Z 264.782,A -85,B 0,C 180,E1 -13825.955,E2 -13825.955} C_VEL
LIN {X 0,Y 347.761,Z 264.786,A -85,B 0,C 180,E1 -13829.652,E2 -13829.652} C_VEL
LIN {X 0,Y 347.849,Z 264.775,A -85,B 0,C 180,E1 -13832.743,E2 -13832.743} C_VEL
LIN {X 0,Y 347.784,Z 264.782,A -85,B 0,C 180,E1 -13836.16,E2 -13836.16} C_VEL
LIN {X 0,Y 347.809,Z 264.778,A -85,B 0,C 180,E1 -13839.908,E2 -13839.908} C_VEL
LIN {X 0,Y 347.861,Z 264.777,A -85,B 0,C 180,E1 -13842.358,E2 -13842.358} C_VEL
LIN {X 0,Y 347.892,Z 264.776,A -85,B 0,C 180,E1 -13845.969,E2 -13845.969} C_VEL
LIN {X 0,Y 347.922,Z 264.768,A -85,B 0,C 180,E1 -13849.524,E2 -13849.524} C_VEL
LIN {X 0,Y 348.086,Z 264.741,A -85,B 0,C 180,E1 -13853.04,E2 -13853.04} C_VEL
LIN {X 0,Y 348.2,Z 264.731,A -85,B 0,C 180,E1 -13857.685,E2 -13857.685} C_VEL
LIN {X 0,Y 348.36,Z 264.713,A -85,B 0,C 180,E1 -13859.998,E2 -13859.998} C_VEL
LIN {X 0,Y 348.2,Z 264.732,A -85,B 0,C 180,E1 -13862.312,E2 -13862.312} C_VEL
LIN {X 0,Y 348.084,Z 264.748,A -85,B 0,C 180,E1 -13866.956,E2 -13866.956} C_VEL
LIN {X 0,Y 347.919,Z 264.765,A -85,B 0,C 180,E1 -13870.473,E2 -13870.473} C_VEL
LIN {X 0,Y 347.888,Z 264.769,A -85,B 0,C 180,E1 -13874.148,E2 -13874.148} C_VEL
LIN {X 0,Y 347.881,Z 264.773,A -85,B 0,C 180,E1 -13878.289,E2 -13878.289} C_VEL
LIN {X 0,Y 347.789,Z 264.786,A -85,B 0,C 180,E1 -13881.639,E2 -13881.639} C_VEL
LIN {X 0,Y 347.806,Z 264.788,A -85,B 0,C 180,E1 -13885.107,E2 -13885.107} C_VEL
LIN {X 0,Y 347.8,Z 264.785,A -85,B 0,C 180,E1 -13887.693,E2 -13887.693} C_VEL
LIN {X 0,Y 347.752,Z 264.776,A -85,B 0,C 180,E1 -13890.345,E2 -13890.345} C_VEL
LIN {X 0,Y 347.731,Z 264.784,A -85,B 0,C 180,E1 -13894.463,E2 -13894.463} C_VEL
LIN {X 0,Y 347.765,Z 264.788,A -85,B 0,C 180,E1 -13897.989,E2 -13897.989} C_VEL
LIN {X 0,Y 347.771,Z 264.784,A -85,B 0,C 180,E1 -13901.825,E2 -13901.825} C_VEL
LIN {X 0,Y 347.823,Z 264.857,A -85,B 0,C 180,E1 -13903.639,E2 -13903.639} C_VEL
LIN {X 0,Y 350.128,Z 273.393,A -85,B 0,C 180,E1 -13906.336,E2 -13906.336} C_VEL
LIN {X 0,Y 360.561,Z 294.385,A -85,B 0,C 180,E1 -13907.943,E2 -13907.943} C_VEL
LIN {X 0,Y 365.452,Z 306.005,A -85,B 0,C 180,E1 -13908.692,E2 -13908.692} C_VEL
LIN {X 0,Y 365.594,Z 310.18,A -85,B 0,C 180,E1 -13908.801,E2 -13908.801} C_VEL
LIN {X 0,Y 362.778,Z 409.721,A -85,B 0,C 180,E1 -13910.829,E2 -13910.829} C_VEL
LIN {X 0,Y 361.891,Z 424.314,A -85,B 0,C 180,E1 -13911.352,E2 -13911.352} C_VEL
LIN {X 0,Y 360.683,Z 437.758,A -85,B 0,C 180,E1 -13912.049,E2 -13912.049} C_VEL
LIN {X 0,Y 359.36,Z 450.643,A -85,B 0,C 180,E1 -13912.953,E2 -13912.953} C_VEL
LIN {X 0,Y 357.73,Z 463.115,A -85,B 0,C 180,E1 -13914.062,E2 -13914.062} C_VEL
LIN {X 0,Y 356.109,Z 474.002,A -85,B 0,C 180,E1 -13915.261,E2 -13915.261} C_VEL
LIN {X 0,Y 354.29,Z 485.22,A -85,B 0,C 180,E1 -13916.772,E2 -13916.772} C_VEL
LIN {X 0,Y 352.503,Z 495.363,A -85,B 0,C 180,E1 -13918.443,E2 -13918.443} C_VEL
LIN {X 0,Y 350.881,Z 504.483,A -85,B 0,C 180,E1 -13920.283,E2 -13920.283} C_VEL
LIN {X 0,Y 349.493,Z 512.306,A -85,B 0,C 180,E1 -13922.222,E2 -13922.222} C_VEL
LIN {X 0,Y 348.302,Z 519.009,A -85,B 0,C 180,E1 -13924.29,E2 -13924.29} C_VEL
LIN {X 0,Y 347.507,Z 523.782,A -85,B 0,C 180,E1 -13926.142,E2 -13926.142} C_VEL
LIN {X 0,Y 346.905,Z 527.536,A -85,B 0,C 180,E1 -13927.989,E2 -13927.989} C_VEL
LIN {X 0,Y 346.484,Z 530.382,A -85,B 0,C 180,E1 -13929.83,E2 -13929.83} C_VEL
LIN {X 0,Y 346.13,Z 532.802,A -85,B 0,C 180,E1 -13932.268,E2 -13932.268} C_VEL
LIN {X 0,Y 345.941,Z 533.782,A -85,B 0,C 180,E1 -13934.687,E2 -13934.687} C_VEL
LIN {X 0,Y 346.012,Z 533.342,A -85,B 0,C 180,E1 -13937.138,E2 -13937.138} C_VEL
LIN {X 0,Y 346.035,Z 531.571,A -85,B 0,C 180,E1 -13939.468,E2 -13939.468} C_VEL
LIN {X 0,Y 346.319,Z 528.376,A -85,B 0,C 180,E1 -13941.834,E2 -13941.834} C_VEL
LIN {X 0,Y 346.602,Z 525.23,A -85,B 0,C 180,E1 -13943.476,E2 -13943.476} C_VEL
LIN {X 0,Y 346.919,Z 520.722,A -85,B 0,C 180,E1 -13945.352,E2 -13945.352} C_VEL
LIN {X 0,Y 347.544,Z 514.512,A -85,B 0,C 180,E1 -13947.392,E2 -13947.392} C_VEL
LIN {X 0,Y 348.511,Z 506.771,A -85,B 0,C 180,E1 -13949.422,E2 -13949.422} C_VEL
LIN {X 0,Y 349.481,Z 498.714,A -85,B 0,C 180,E1 -13951.152,E2 -13951.152} C_VEL
LIN {X 0,Y 350.72,Z 489.004,A -85,B 0,C 180,E1 -13952.872,E2 -13952.872} C_VEL
LIN {X 0,Y 352.102,Z 478.227,A -85,B 0,C 180,E1 -13954.436,E2 -13954.436} C_VEL
LIN {X 0,Y 353.497,Z 466.484,A -85,B 0,C 180,E1 -13955.827,E2 -13955.827} C_VEL
LIN {X 0,Y 354.636,Z 454.601,A -85,B 0,C 180,E1 -13956.972,E2 -13956.972} C_VEL
LIN {X 0,Y 355.786,Z 441.809,A -85,B 0,C 180,E1 -13957.948,E2 -13957.948} C_VEL
LIN {X 0,Y 356.708,Z 428.748,A -85,B 0,C 180,E1 -13958.712,E2 -13958.712} C_VEL
LIN {X 0,Y 357.412,Z 414.66,A -85,B 0,C 180,E1 -13959.3,E2 -13959.3} C_VEL
LIN {X 0,Y 357.879,Z 398.253,A -85,B 0,C 180,E1 -13959.716,E2 -13959.716} C_VEL
LIN {X 0,Y 359.783,Z 311.326,A -85,B 0,C 180,E1 -13961.444,E2 -13961.444} C_VEL
LIN {X 0,Y 359.033,Z 307.588,A -85,B 0,C 180,E1 -13961.572,E2 -13961.572} C_VEL
LIN {X 0,Y 357.255,Z 304.226,A -85,B 0,C 180,E1 -13961.759,E2 -13961.759} C_VEL
LIN {X 0,Y 351.258,Z 295.788,A -85,B 0,C 180,E1 -13962.341,E2 -13962.341} C_VEL
LIN {X 0,Y 350.23,Z 293.368,A -85,B 0,C 180,E1 -13962.464,E2 -13962.464} C_VEL
LIN {X 0,Y 342.392,Z 272.633,A -85,B 0,C 180,E1 -13963.502,E2 -13963.502} C_VEL
LIN {X 0,Y 340.798,Z 265.66,A -85,B 0,C 180,E1 -13965.479,E2 -13965.479} C_VEL
LIN {X 0,Y 340.826,Z 265.654,A -85,B 0,C 180,E1 -13968.468,E2 -13968.468} C_VEL
LIN {X 0,Y 340.741,Z 265.668,A -85,B 0,C 180,E1 -13971.857,E2 -13971.857} C_VEL
LIN {X 0,Y 340.76,Z 265.665,A -85,B 0,C 180,E1 -13975.665,E2 -13975.665} C_VEL
LIN {X 0,Y 340.73,Z 265.664,A -85,B 0,C 180,E1 -13978.32,E2 -13978.32} C_VEL
LIN {X 0,Y 340.692,Z 265.67,A -85,B 0,C 180,E1 -13981.045,E2 -13981.045} C_VEL
LIN {X 0,Y 340.706,Z 265.671,A -85,B 0,C 180,E1 -13985.28,E2 -13985.28} C_VEL
LIN {X 0,Y 340.707,Z 265.667,A -85,B 0,C 180,E1 -13988.389,E2 -13988.389} C_VEL
LIN {X 0,Y 340.714,Z 265.67,A -85,B 0,C 180,E1 -13991.305,E2 -13991.305} C_VEL
LIN {X 0,Y 340.769,Z 265.659,A -85,B 0,C 180,E1 -13994.523,E2 -13994.523} C_VEL
LIN {X 0,Y 340.74,Z 265.662,A -85,B 0,C 180,E1 -13997.946,E2 -13997.946} C_VEL
LIN {X 0,Y 340.723,Z 265.665,A -85,B 0,C 180,E1 -14000.253,E2 -14000.253} C_VEL
LIN {X 0,Y 340.699,Z 265.667,A -85,B 0,C 180,E1 -14003.56,E2 -14003.56} C_VEL
LIN {X 0,Y 340.681,Z 265.669,A -85,B 0,C 180,E1 -14006.155,E2 -14006.155} C_VEL
LIN {X 0,Y 340.764,Z 265.66,A -85,B 0,C 180,E1 -14010.334,E2 -14010.334} C_VEL
LIN {X 0,Y 340.795,Z 265.658,A -85,B 0,C 180,E1 -14013.021,E2 -14013.021} C_VEL
LIN {X 0,Y 340.719,Z 265.671,A -85,B 0,C 180,E1 -14016.928,E2 -14016.928} C_VEL
LIN {X 0,Y 340.781,Z 265.662,A -85,B 0,C 180,E1 -14020.735,E2 -14020.735} C_VEL
LIN {X 0,Y 340.777,Z 265.66,A -85,B 0,C 180,E1 -14023.22,E2 -14023.22} C_VEL
LIN {X 0,Y 340.835,Z 265.655,A -85,B 0,C 180,E1 -14026.892,E2 -14026.892} C_VEL
LIN {X 0,Y 340.906,Z 265.646,A -85,B 0,C 180,E1 -14030.509,E2 -14030.509} C_VEL
LIN {X 0,Y 341.052,Z 265.624,A -85,B 0,C 180,E1 -14032.899,E2 -14032.899} C_VEL
LIN {X 0,Y 341.163,Z 265.61,A -85,B 0,C 180,E1 -14037.64,E2 -14037.64} C_VEL
LIN {X 0,Y 341.289,Z 265.596,A -85,B 0,C 180,E1 -14040.002,E2 -14040.002} C_VEL
LIN {X 0,Y 341.164,Z 265.613,A -85,B 0,C 180,E1 -14042.363,E2 -14042.363} C_VEL
LIN {X 0,Y 341.054,Z 265.624,A -85,B 0,C 180,E1 -14047.104,E2 -14047.104} C_VEL
LIN {X 0,Y 340.866,Z 265.647,A -85,B 0,C 180,E1 -14050.695,E2 -14050.695} C_VEL
LIN {X 0,Y 340.859,Z 265.652,A -85,B 0,C 180,E1 -14054.326,E2 -14054.326} C_VEL
LIN {X 0,Y 340.834,Z 265.653,A -85,B 0,C 180,E1 -14058.468,E2 -14058.468} C_VEL
LIN {X 0,Y 340.715,Z 265.669,A -85,B 0,C 180,E1 -14061.843,E2 -14061.843} C_VEL
LIN {X 0,Y 340.77,Z 265.662,A -85,B 0,C 180,E1 -14065.666,E2 -14065.666} C_VEL
LIN {X 0,Y 340.74,Z 265.665,A -85,B 0,C 180,E1 -14068.321,E2 -14068.321} C_VEL
LIN {X 0,Y 340.714,Z 265.666,A -85,B 0,C 180,E1 -14071.044,E2 -14071.044} C_VEL
LIN {X 0,Y 340.718,Z 265.667,A -85,B 0,C 180,E1 -14075.28,E2 -14075.28} C_VEL
LIN {X 0,Y 340.71,Z 265.668,A -85,B 0,C 180,E1 -14078.387,E2 -14078.387} C_VEL
LIN {X 0,Y 340.699,Z 265.671,A -85,B 0,C 180,E1 -14082.047,E2 -14082.047} C_VEL
LIN {X 0,Y 340.653,Z 265.675,A -85,B 0,C 180,E1 -14086.228,E2 -14086.228} C_VEL
LIN {X 0,Y 340.69,Z 265.674,A -85,B 0,C 180,E1 -14089.754,E2 -14089.754} C_VEL
LIN {X 0,Y 340.707,Z 265.671,A -85,B 0,C 180,E1 -14093.259,E2 -14093.259} C_VEL
LIN {X 0,Y 340.741,Z 265.784,A -85,B 0,C 180,E1 -14096.825,E2 -14096.825} C_VEL
LIN {X 0,Y 343.833,Z 279.419,A -85,B 0,C 180,E1 -14100.29,E2 -14100.29} C_VEL
LIN {X 0,Y 345.94,Z 289.751,A -85,B 0,C 180,E1 -14102.787,E2 -14102.787} C_VEL
LIN {X 0,Y 347.572,Z 297.589,A -85,B 0,C 180,E1 -14103.075,E2 -14103.075} C_VEL
LIN {X 0,Y 352.883,Z 331.191,A -85,B 0,C 180,E1 -14104.169,E2 -14104.169} C_VEL
LIN {X 0,Y 350.784,Z 427.281,A -85,B 0,C 180,E1 -14106.143,E2 -14106.143} C_VEL
LIN {X 0,Y 350.058,Z 441.399,A -85,B 0,C 180,E1 -14106.64,E2 -14106.64} C_VEL
LIN {X 0,Y 349.004,Z 455.134,A -85,B 0,C 180,E1 -14107.349,E2 -14107.349} C_VEL
LIN {X 0,Y 347.873,Z 467.609,A -85,B 0,C 180,E1 -14108.21,E2 -14108.21} C_VEL
LIN {X 0,Y 346.48,Z 480.638,A -85,B 0,C 180,E1 -14109.364,E2 -14109.364} C_VEL
LIN {X 0,Y 345.086,Z 492.469,A -85,B 0,C 180,E1 -14110.674,E2 -14110.674} C_VEL
LIN {X 0,Y 343.689,Z 503.281,A -85,B 0,C 180,E1 -14112.138,E2 -14112.138} C_VEL
LIN {X 0,Y 342.307,Z 513.984,A -85,B 0,C 180,E1 -14113.909,E2 -14113.909} C_VEL
LIN {X 0,Y 341.335,Z 522.814,A -85,B 0,C 180,E1 -14115.696,E2 -14115.696} C_VEL
LIN {X 0,Y 340.37,Z 531.256,A -85,B 0,C 180,E1 -14117.781,E2 -14117.781} C_VEL
LIN {X 0,Y 339.673,Z 538.016,A -85,B 0,C 180,E1 -14119.871,E2 -14119.871} C_VEL
LIN {X 0,Y 339.336,Z 542.662,A -85,B 0,C 180,E1 -14121.664,E2 -14121.664} C_VEL
LIN {X 0,Y 339.169,Z 546.374,A -85,B 0,C 180,E1 -14123.456,E2 -14123.456} C_VEL
LIN {X 0,Y 339.042,Z 549.255,A -85,B 0,C 180,E1 -14125.244,E2 -14125.244} C_VEL
LIN {X 0,Y 339.054,Z 550.695,A -85,B 0,C 180,E1 -14126.435,E2 -14126.435} C_VEL
LIN {X 0,Y 339.024,Z 552.528,A -85,B 0,C 180,E1 -14128.812,E2 -14128.812} C_VEL
LIN {X 0,Y 339.068,Z 552.938,A -85,B 0,C 180,E1 -14130,E2 -14130} C_VEL
LIN {X 0,Y 338.993,Z 552.751,A -85,B 0,C 180,E1 -14132.376,E2 -14132.376} C_VEL
LIN {X 0,Y 339.048,Z 551.236,A -85,B 0,C 180,E1 -14134.756,E2 -14134.756} C_VEL
LIN {X 0,Y 339.25,Z 548.365,A -85,B 0,C 180,E1 -14137.14,E2 -14137.14} C_VEL
LIN {X 0,Y 339.683,Z 544.066,A -85,B 0,C 180,E1 -14139.527,E2 -14139.527} C_VEL
LIN {X 0,Y 340.465,Z 538.223,A -85,B 0,C 180,E1 -14141.912,E2 -14141.912} C_VEL
LIN {X 0,Y 341.608,Z 531.673,A -85,B 0,C 180,E1 -14143.989,E2 -14143.989} C_VEL
LIN {X 0,Y 342.96,Z 523.589,A -85,B 0,C 180,E1 -14146.06,E2 -14146.06} C_VEL
LIN {X 0,Y 344.507,Z 515.154,A -85,B 0,C 180,E1 -14147.818,E2 -14147.818} C_VEL
LIN {X 0,Y 346.43,Z 505.006,A -85,B 0,C 180,E1 -14149.556,E2 -14149.556} C_VEL
LIN {X 0,Y 348.419,Z 493.677,A -85,B 0,C 180,E1 -14151.134,E2 -14151.134} C_VEL
LIN {X 0,Y 350.34,Z 481.513,A -85,B 0,C 180,E1 -14152.508,E2 -14152.508} C_VEL
LIN {X 0,Y 352.221,Z 468.47,A -85,B 0,C 180,E1 -14153.675,E2 -14153.675} C_VEL
LIN {X 0,Y 353.8,Z 455.515,A -85,B 0,C 180,E1 -14154.576,E2 -14154.576} C_VEL
LIN {X 0,Y 355.179,Z 441.604,A -85,B 0,C 180,E1 -14155.294,E2 -14155.294} C_VEL
LIN {X 0,Y 356.233,Z 427.041,A -85,B 0,C 180,E1 -14155.801,E2 -14155.801} C_VEL
LIN {X 0,Y 358.915,Z 331.974,A -85,B 0,C 180,E1 -14157.775,E2 -14157.775} C_VEL
LIN {X 0,Y 354.371,Z 308.308,A -85,B 0,C 180,E1 -14158.794,E2 -14158.794} C_VEL
LIN {X 0,Y 352.94,Z 302.587,A -85,B 0,C 180,E1 -14159.081,E2 -14159.081} C_VEL
LIN {X 0,Y 348.229,Z 292.339,A -85,B 0,C 180,E1 -14159.84,E2 -14159.84} C_VEL
LIN {X 0,Y 346.681,Z 288.857,A -85,B 0,C 180,E1 -14160.129,E2 -14160.129} C_VEL
LIN {X 0,Y 344.595,Z 280.081,A -85,B 0,C 180,E1 -14162.591,E2 -14162.591} C_VEL
LIN {X 0,Y 341.974,Z 270.246,A -85,B 0,C 180,E1 -14165.54,E2 -14165.54} C_VEL
LIN {X 0,Y 340.725,Z 265.667,A -85,B 0,C 180,E1 -14167.015,E2 -14167.015} C_VEL
LIN {X 0,Y 340.765,Z 265.656,A -85,B 0,C 180,E1 -14170.261,E2 -14170.261} C_VEL
LIN {X 0,Y 340.717,Z 265.668,A -85,B 0,C 180,E1 -14173.783,E2 -14173.783} C_VEL
LIN {X 0,Y 340.678,Z 265.673,A -85,B 0,C 180,E1 -14177.095,E2 -14177.095} C_VEL
LIN {X 0,Y 340.698,Z 265.668,A -85,B 0,C 180,E1 -14180.246,E2 -14180.246} C_VEL
LIN {X 0,Y 340.708,Z 265.649,A -85,B 0,C 180,E1 -14183.558,E2 -14183.558} C_VEL
LIN {X 0,Y 340.69,Z 265.663,A -85,B 0,C 180,E1 -14186.152,E2 -14186.152} C_VEL
LIN {X 0,Y 340.772,Z 265.663,A -85,B 0,C 180,E1 -14190.331,E2 -14190.331} C_VEL
LIN {X 0,Y 340.802,Z 265.653,A -85,B 0,C 180,E1 -14193.018,E2 -14193.018} C_VEL
LIN {X 0,Y 340.724,Z 265.664,A -85,B 0,C 180,E1 -14196.925,E2 -14196.925} C_VEL
LIN {X 0,Y 340.787,Z 265.655,A -85,B 0,C 180,E1 -14200.732,E2 -14200.732} C_VEL
LIN {X 0,Y 340.781,Z 265.657,A -85,B 0,C 180,E1 -14203.217,E2 -14203.217} C_VEL
LIN {X 0,Y 340.838,Z 265.653,A -85,B 0,C 180,E1 -14206.889,E2 -14206.889} C_VEL
LIN {X 0,Y 340.92,Z 265.643,A -85,B 0,C 180,E1 -14210.506,E2 -14210.506} C_VEL
LIN {X 0,Y 341.054,Z 265.616,A -85,B 0,C 180,E1 -14212.896,E2 -14212.896} C_VEL
LIN {X 0,Y 341.162,Z 265.607,A -85,B 0,C 180,E1 -14217.637,E2 -14217.637} C_VEL
LIN {X 0,Y 341.309,Z 265.592,A -85,B 0,C 180,E1 -14219.998,E2 -14219.998} C_VEL
LIN {X 0,Y 341.161,Z 265.609,A -85,B 0,C 180,E1 -14222.36,E2 -14222.36} C_VEL
LIN {X 0,Y 341.052,Z 265.626,A -85,B 0,C 180,E1 -14227.101,E2 -14227.101} C_VEL
LIN {X 0,Y 340.861,Z 265.645,A -85,B 0,C 180,E1 -14230.692,E2 -14230.692} C_VEL
LIN {X 0,Y 340.853,Z 265.645,A -85,B 0,C 180,E1 -14234.323,E2 -14234.323} C_VEL
LIN {X 0,Y 340.828,Z 265.652,A -85,B 0,C 180,E1 -14238.466,E2 -14238.466} C_VEL
LIN {X 0,Y 340.743,Z 265.664,A -85,B 0,C 180,E1 -14241.856,E2 -14241.856} C_VEL
LIN {X 0,Y 340.764,Z 265.663,A -85,B 0,C 180,E1 -14245.663,E2 -14245.663} C_VEL
LIN {X 0,Y 340.73,Z 265.669,A -85,B 0,C 180,E1 -14248.318,E2 -14248.318} C_VEL
LIN {X 0,Y 340.691,Z 265.654,A -85,B 0,C 180,E1 -14251.043,E2 -14251.043} C_VEL
LIN {X 0,Y 340.706,Z 265.656,A -85,B 0,C 180,E1 -14255.278,E2 -14255.278} C_VEL
LIN {X 0,Y 340.702,Z 265.663,A -85,B 0,C 180,E1 -14258.386,E2 -14258.386} C_VEL
LIN {X 0,Y 340.713,Z 265.667,A -85,B 0,C 180,E1 -14261.303,E2 -14261.303} C_VEL
LIN {X 0,Y 340.753,Z 265.754,A -85,B 0,C 180,E1 -14262.941,E2 -14262.941} C_VEL
LIN {X 0,Y 342.961,Z 273.723,A -85,B 0,C 180,E1 -14265.526,E2 -14265.526} C_VEL
LIN {X 0,Y 352.603,Z 292.536,A -85,B 0,C 180,E1 -14267.072,E2 -14267.072} C_VEL
LIN {X 0,Y 359.584,Z 308.254,A -85,B 0,C 180,E1 -14268.169,E2 -14268.169} C_VEL
LIN {X 0,Y 356.578,Z 410.294,A -85,B 0,C 180,E1 -14270.286,E2 -14270.286} C_VEL
LIN {X 0,Y 355.713,Z 424.096,A -85,B 0,C 180,E1 -14270.786,E2 -14270.786} C_VEL
LIN {X 0,Y 354.393,Z 438.164,A -85,B 0,C 180,E1 -14271.524,E2 -14271.524} C_VEL
LIN {X 0,Y 353.063,Z 450.592,A -85,B 0,C 180,E1 -14272.408,E2 -14272.408} C_VEL
LIN {X 0,Y 351.441,Z 462.695,A -85,B 0,C 180,E1 -14273.493,E2 -14273.493} C_VEL
LIN {X 0,Y 349.534,Z 474.927,A -85,B 0,C 180,E1 -14274.862,E2 -14274.862} C_VEL
LIN {X 0,Y 347.72,Z 485.481,A -85,B 0,C 180,E1 -14276.317,E2 -14276.317} C_VEL
LIN {X 0,Y 345.752,Z 496.06,A -85,B 0,C 180,E1 -14278.097,E2 -14278.097} C_VEL
LIN {X 0,Y 344.072,Z 505.087,A -85,B 0,C 180,E1 -14279.972,E2 -14279.972} C_VEL
LIN {X 0,Y 342.657,Z 512.555,A -85,B 0,C 180,E1 -14281.873,E2 -14281.873} C_VEL
LIN {X 0,Y 341.516,Z 518.54,A -85,B 0,C 180,E1 -14283.741,E2 -14283.741} C_VEL
LIN {X 0,Y 340.638,Z 523.444,A -85,B 0,C 180,E1 -14285.63,E2 -14285.63} C_VEL
LIN {X 0,Y 339.946,Z 527.336,A -85,B 0,C 180,E1 -14287.514,E2 -14287.514} C_VEL
LIN {X 0,Y 339.493,Z 530.308,A -85,B 0,C 180,E1 -14289.396,E2 -14289.396} C_VEL
LIN {X 0,Y 339.072,Z 532.856,A -85,B 0,C 180,E1 -14291.887,E2 -14291.887} C_VEL
LIN {X 0,Y 338.849,Z 533.956,A -85,B 0,C 180,E1 -14294.358,E2 -14294.358} C_VEL
LIN {X 0,Y 338.913,Z 533.653,A -85,B 0,C 180,E1 -14296.815,E2 -14296.815} C_VEL
LIN {X 0,Y 338.948,Z 531.977,A -85,B 0,C 180,E1 -14299.245,E2 -14299.245} C_VEL
LIN {X 0,Y 339.196,Z 528.904,A -85,B 0,C 180,E1 -14301.661,E2 -14301.661} C_VEL
LIN {X 0,Y 339.621,Z 524.37,A -85,B 0,C 180,E1 -14304.061,E2 -14304.061} C_VEL
LIN {X 0,Y 339.994,Z 519.883,A -85,B 0,C 180,E1 -14305.851,E2 -14305.851} C_VEL
LIN {X 0,Y 340.667,Z 513.421,A -85,B 0,C 180,E1 -14307.931,E2 -14307.931} C_VEL
LIN {X 0,Y 341.718,Z 505.397,A -85,B 0,C 180,E1 -14310,E2 -14310} C_VEL
LIN {X 0,Y 342.832,Z 497.009,A -85,B 0,C 180,E1 -14311.762,E2 -14311.762} C_VEL
LIN {X 0,Y 344.126,Z 486.922,A -85,B 0,C 180,E1 -14313.513,E2 -14313.513} C_VEL
LIN {X 0,Y 345.601,Z 475.608,A -85,B 0,C 180,E1 -14315.105,E2 -14315.105} C_VEL
LIN {X 0,Y 346.906,Z 464.303,A -85,B 0,C 180,E1 -14316.407,E2 -14316.407} C_VEL
LIN {X 0,Y 348.146,Z 452.164,A -85,B 0,C 180,E1 -14317.54,E2 -14317.54} C_VEL
LIN {X 0,Y 349.287,Z 438.584,A -85,B 0,C 180,E1 -14318.534,E2 -14318.534} C_VEL
LIN {X 0,Y 350.256,Z 424.278,A -85,B 0,C 180,E1 -14319.31,E2 -14319.31} C_VEL
LIN {X 0,Y 350.868,Z 410.102,A -85,B 0,C 180,E1 -14319.839,E2 -14319.839} C_VEL
LIN {X 0,Y 352.545,Z 341.733,A -85,B 0,C 180,E1 -14321.254,E2 -14321.254} C_VEL
LIN {X 0,Y 353.332,Z 305.391,A -85,B 0,C 180,E1 -14321.992,E2 -14321.992} C_VEL
LIN {X 0,Y 351.124,Z 295.828,A -85,B 0,C 180,E1 -14322.349,E2 -14322.349} C_VEL
LIN {X 0,Y 350.23,Z 293.368,A -85,B 0,C 180,E1 -14322.464,E2 -14322.464} C_VEL
LIN {X 0,Y 348.473,Z 290.04,A -85,B 0,C 180,E1 -14322.66,E2 -14322.66} C_VEL
LIN {X 0,Y 344.059,Z 285.652,A -85,B 0,C 180,E1 -14323.069,E2 -14323.069} C_VEL
LIN {X 0,Y 339.41,Z 281.397,A -85,B 0,C 180,E1 -14323.502,E2 -14323.502} C_VEL
LIN {X 0,Y 337.302,Z 278.239,A -85,B 0,C 180,E1 -14323.73,E2 -14323.73} C_VEL
LIN {X 0,Y 335.181,Z 272.842,A -85,B 0,C 180,E1 -14324.035,E2 -14324.035} C_VEL
LIN {X 0,Y 333.765,Z 266.535,A -85,B 0,C 180,E1 -14325.887,E2 -14325.887} C_VEL
LIN {X 0,Y 333.785,Z 266.531,A -85,B 0,C 180,E1 -14328.656,E2 -14328.656} C_VEL
LIN {X 0,Y 333.68,Z 266.544,A -85,B 0,C 180,E1 -14332.279,E2 -14332.279} C_VEL
LIN {X 0,Y 333.723,Z 266.538,A -85,B 0,C 180,E1 -14336.247,E2 -14336.247} C_VEL
LIN {X 0,Y 333.699,Z 266.54,A -85,B 0,C 180,E1 -14338.973,E2 -14338.973} C_VEL
LIN {X 0,Y 333.631,Z 266.548,A -85,B 0,C 180,E1 -14342.588,E2 -14342.588} C_VEL
LIN {X 0,Y 333.665,Z 266.544,A -85,B 0,C 180,E1 -14346.14,E2 -14346.14} C_VEL
LIN {X 0,Y 333.672,Z 266.547,A -85,B 0,C 180,E1 -14349.188,E2 -14349.188} C_VEL
LIN {X 0,Y 333.691,Z 266.541,A -85,B 0,C 180,E1 -14352.514,E2 -14352.514} C_VEL
LIN {X 0,Y 333.717,Z 266.536,A -85,B 0,C 180,E1 -14355.978,E2 -14355.978} C_VEL
LIN {X 0,Y 333.69,Z 266.546,A -85,B 0,C 180,E1 -14359.306,E2 -14359.306} C_VEL
LIN {X 0,Y 333.654,Z 266.547,A -85,B 0,C 180,E1 -14363.169,E2 -14363.169} C_VEL
LIN {X 0,Y 333.626,Z 266.55,A -85,B 0,C 180,E1 -14366.793,E2 -14366.793} C_VEL
LIN {X 0,Y 333.692,Z 266.541,A -85,B 0,C 180,E1 -14369.712,E2 -14369.712} C_VEL
LIN {X 0,Y 333.734,Z 266.534,A -85,B 0,C 180,E1 -14372.403,E2 -14372.403} C_VEL
LIN {X 0,Y 333.717,Z 266.541,A -85,B 0,C 180,E1 -14375.092,E2 -14375.092} C_VEL
LIN {X 0,Y 333.675,Z 266.547,A -85,B 0,C 180,E1 -14379.021,E2 -14379.021} C_VEL
LIN {X 0,Y 333.784,Z 266.529,A -85,B 0,C 180,E1 -14381.591,E2 -14381.591} C_VEL
LIN {X 0,Y 333.8,Z 266.526,A -85,B 0,C 180,E1 -14385.578,E2 -14385.578} C_VEL
LIN {X 0,Y 333.825,Z 266.526,A -85,B 0,C 180,E1 -14389.08,E2 -14389.08} C_VEL
LIN {X 0,Y 333.999,Z 266.503,A -85,B 0,C 180,E1 -14392.749,E2 -14392.749} C_VEL
LIN {X 0,Y 333.804,Z 266.526,A -85,B 0,C 180,E1 -14395.171,E2 -14395.171} C_VEL
LIN {X 0,Y 334.101,Z 266.49,A -85,B 0,C 180,E1 -14397.59,E2 -14397.59} C_VEL
LIN {X 0,Y 334.24,Z 266.474,A -85,B 0,C 180,E1 -14400.002,E2 -14400.002} C_VEL
LIN {X 0,Y 334.101,Z 266.491,A -85,B 0,C 180,E1 -14402.413,E2 -14402.413} C_VEL
LIN {X 0,Y 334.01,Z 266.503,A -85,B 0,C 180,E1 -14406.041,E2 -14406.041} C_VEL
LIN {X 0,Y 333.954,Z 266.512,A -85,B 0,C 180,E1 -14408.473,E2 -14408.473} C_VEL
LIN {X 0,Y 333.787,Z 266.531,A -85,B 0,C 180,E1 -14412.156,E2 -14412.156} C_VEL
LIN {X 0,Y 333.775,Z 266.533,A -85,B 0,C 180,E1 -14415.888,E2 -14415.888} C_VEL
LIN {X 0,Y 333.793,Z 266.529,A -85,B 0,C 180,E1 -14418.656,E2 -14418.656} C_VEL
LIN {X 0,Y 333.654,Z 266.549,A -85,B 0,C 180,E1 -14422.282,E2 -14422.282} C_VEL
LIN {X 0,Y 333.734,Z 266.539,A -85,B 0,C 180,E1 -14426.248,E2 -14426.248} C_VEL
LIN {X 0,Y 333.71,Z 266.539,A -85,B 0,C 180,E1 -14428.974,E2 -14428.974} C_VEL
LIN {X 0,Y 333.65,Z 266.547,A -85,B 0,C 180,E1 -14432.591,E2 -14432.591} C_VEL
LIN {X 0,Y 333.676,Z 266.546,A -85,B 0,C 180,E1 -14436.14,E2 -14436.14} C_VEL
LIN {X 0,Y 333.647,Z 266.548,A -85,B 0,C 180,E1 -14439.194,E2 -14439.194} C_VEL
LIN {X 0,Y 333.633,Z 266.548,A -85,B 0,C 180,E1 -14442.501,E2 -14442.501} C_VEL
LIN {X 0,Y 333.597,Z 266.556,A -85,B 0,C 180,E1 -14445.956,E2 -14445.956} C_VEL
LIN {X 0,Y 333.649,Z 266.55,A -85,B 0,C 180,E1 -14449.317,E2 -14449.317} C_VEL
LIN {X 0,Y 333.667,Z 266.548,A -85,B 0,C 180,E1 -14453.169,E2 -14453.169} C_VEL
LIN {X 0,Y 333.705,Z 266.727,A -85,B 0,C 180,E1 -14456.439,E2 -14456.439} C_VEL
LIN {X 0,Y 336.753,Z 280.184,A -85,B 0,C 180,E1 -14459.943,E2 -14459.943} C_VEL
LIN {X 0,Y 338.714,Z 289.543,A -85,B 0,C 180,E1 -14462.263,E2 -14462.263} C_VEL
LIN {X 0,Y 340.571,Z 295.898,A -85,B 0,C 180,E1 -14462.543,E2 -14462.543} C_VEL
LIN {X 0,Y 346.29,Z 332.025,A -85,B 0,C 180,E1 -14463.752,E2 -14463.752} C_VEL
LIN {X 0,Y 344.135,Z 426.757,A -85,B 0,C 180,E1 -14465.733,E2 -14465.733} C_VEL
LIN {X 0,Y 343.39,Z 441.022,A -85,B 0,C 180,E1 -14466.239,E2 -14466.239} C_VEL
LIN {X 0,Y 342.305,Z 454.811,A -85,B 0,C 180,E1 -14466.96,E2 -14466.96} C_VEL
LIN {X 0,Y 341.153,Z 467.111,A -85,B 0,C 180,E1 -14467.819,E2 -14467.819} C_VEL
LIN {X 0,Y 339.79,Z 479.784,A -85,B 0,C 180,E1 -14468.953,E2 -14468.953} C_VEL
LIN {X 0,Y 338.44,Z 490.433,A -85,B 0,C 180,E1 -14470.121,E2 -14470.121} C_VEL
LIN {X 0,Y 337.184,Z 500.58,A -85,B 0,C 180,E1 -14471.467,E2 -14471.467} C_VEL
LIN {X 0,Y 335.642,Z 511.7,A -85,B 0,C 180,E1 -14473.267,E2 -14473.267} C_VEL
LIN {X 0,Y 334.477,Z 521.131,A -85,B 0,C 180,E1 -14475.141,E2 -14475.141} C_VEL
LIN {X 0,Y 333.589,Z 528.503,A -85,B 0,C 180,E1 -14476.91,E2 -14476.91} C_VEL
LIN {X 0,Y 332.767,Z 535.765,A -85,B 0,C 180,E1 -14479.043,E2 -14479.043} C_VEL
LIN {X 0,Y 332.377,Z 540.833,A -85,B 0,C 180,E1 -14480.875,E2 -14480.875} C_VEL
LIN {X 0,Y 332.101,Z 546.037,A -85,B 0,C 180,E1 -14483.316,E2 -14483.316} C_VEL
LIN {X 0,Y 331.95,Z 548.949,A -85,B 0,C 180,E1 -14485.142,E2 -14485.142} C_VEL
LIN {X 0,Y 331.979,Z 550.419,A -85,B 0,C 180,E1 -14486.359,E2 -14486.359} C_VEL
LIN {X 0,Y 331.929,Z 552.297,A -85,B 0,C 180,E1 -14488.787,E2 -14488.787} C_VEL
LIN {X 0,Y 331.971,Z 552.728,A -85,B 0,C 180,E1 -14490,E2 -14490} C_VEL
LIN {X 0,Y 331.91,Z 552.582,A -85,B 0,C 180,E1 -14492.427,E2 -14492.427} C_VEL
LIN {X 0,Y 331.958,Z 551.107,A -85,B 0,C 180,E1 -14494.858,E2 -14494.858} C_VEL
LIN {X 0,Y 332.174,Z 548.278,A -85,B 0,C 180,E1 -14497.293,E2 -14497.293} C_VEL
LIN {X 0,Y 332.658,Z 544.029,A -85,B 0,C 180,E1 -14499.73,E2 -14499.73} C_VEL
LIN {X 0,Y 333.505,Z 538.24,A -85,B 0,C 180,E1 -14502.165,E2 -14502.165} C_VEL
LIN {X 0,Y 334.654,Z 531.749,A -85,B 0,C 180,E1 -14504.285,E2 -14504.285} C_VEL
LIN {X 0,Y 336.109,Z 523.728,A -85,B 0,C 180,E1 -14506.396,E2 -14506.396} C_VEL
LIN {X 0,Y 337.752,Z 515.36,A -85,B 0,C 180,E1 -14508.187,E2 -14508.187} C_VEL
LIN {X 0,Y 339.765,Z 505.314,A -85,B 0,C 180,E1 -14509.956,E2 -14509.956} C_VEL
LIN {X 0,Y 341.834,Z 494.117,A -85,B 0,C 180,E1 -14511.561,E2 -14511.561} C_VEL
LIN {X 0,Y 343.903,Z 481.531,A -85,B 0,C 180,E1 -14513.016,E2 -14513.016} C_VEL
LIN {X 0,Y 345.766,Z 469.239,A -85,B 0,C 180,E1 -14514.145,E2 -14514.145} C_VEL
LIN {X 0,Y 347.549,Z 455.447,A -85,B 0,C 180,E1 -14515.128,E2 -14515.128} C_VEL
LIN {X 0,Y 348.976,Z 441.599,A -85,B 0,C 180,E1 -14515.857,E2 -14515.857} C_VEL
LIN {X 0,Y 350.064,Z 427.17,A -85,B 0,C 180,E1 -14516.371,E2 -14516.371} C_VEL
LIN {X 0,Y 352.87,Z 333.057,A -85,B 0,C 180,E1 -14518.359,E2 -14518.359} C_VEL
LIN {X 0,Y 348.234,Z 308.991,A -85,B 0,C 180,E1 -14519.43,E2 -14519.43} C_VEL
LIN {X 0,Y 347.033,Z 304.79,A -85,B 0,C 180,E1 -14519.665,E2 -14519.665} C_VEL
LIN {X 0,Y 340.442,Z 291.036,A -85,B 0,C 180,E1 -14520.761,E2 -14520.761} C_VEL
LIN {X 0,Y 339.431,Z 288.588,A -85,B 0,C 180,E1 -14520.977,E2 -14520.977} C_VEL
LIN {X 0,Y 337.103,Z 279.081,A -85,B 0,C 180,E1 -14523.764,E2 -14523.764} C_VEL
LIN {X 0,Y 334.595,Z 269.906,A -85,B 0,C 180,E1 -14526.639,E2 -14526.639} C_VEL
LIN {X 0,Y 333.688,Z 266.541,A -85,B 0,C 180,E1 -14527.74,E2 -14527.74} C_VEL
LIN {X 0,Y 333.7,Z 266.534,A -85,B 0,C 180,E1 -14530.758,E2 -14530.758} C_VEL
LIN {X 0,Y 333.668,Z 266.548,A -85,B 0,C 180,E1 -14534.262,E2 -14534.262} C_VEL
LIN {X 0,Y 333.642,Z 266.548,A -85,B 0,C 180,E1 -14537.617,E2 -14537.617} C_VEL
LIN {X 0,Y 333.651,Z 266.548,A -85,B 0,C 180,E1 -14541.201,E2 -14541.201} C_VEL
LIN {X 0,Y 333.674,Z 266.522,A -85,B 0,C 180,E1 -14543.859,E2 -14543.859} C_VEL
LIN {X 0,Y 333.641,Z 266.55,A -85,B 0,C 180,E1 -14547.411,E2 -14547.411} C_VEL
LIN {X 0,Y 333.709,Z 266.541,A -85,B 0,C 180,E1 -14551.026,E2 -14551.026} C_VEL
LIN {X 0,Y 333.732,Z 266.538,A -85,B 0,C 180,E1 -14553.752,E2 -14553.752} C_VEL
LIN {X 0,Y 333.716,Z 266.543,A -85,B 0,C 180,E1 -14557.912,E2 -14557.912} C_VEL
LIN {X 0,Y 333.789,Z 266.532,A -85,B 0,C 180,E1 -14561.588,E2 -14561.588} C_VEL
LIN {X 0,Y 333.803,Z 266.529,A -85,B 0,C 180,E1 -14565.575,E2 -14565.575} C_VEL
LIN {X 0,Y 333.827,Z 266.519,A -85,B 0,C 180,E1 -14569.076,E2 -14569.076} C_VEL
LIN {X 0,Y 334.006,Z 266.494,A -85,B 0,C 180,E1 -14572.746,E2 -14572.746} C_VEL
LIN {X 0,Y 333.804,Z 266.532,A -85,B 0,C 180,E1 -14575.167,E2 -14575.167} C_VEL
LIN {X 0,Y 334.099,Z 266.486,A -85,B 0,C 180,E1 -14577.587,E2 -14577.587} C_VEL
LIN {X 0,Y 334.259,Z 266.47,A -85,B 0,C 180,E1 -14579.998,E2 -14579.998} C_VEL
LIN {X 0,Y 334.099,Z 266.488,A -85,B 0,C 180,E1 -14582.41,E2 -14582.41} C_VEL
LIN {X 0,Y 333.986,Z 266.501,A -85,B 0,C 180,E1 -14586.674,E2 -14586.674} C_VEL
LIN {X 0,Y 333.851,Z 266.515,A -85,B 0,C 180,E1 -14589.694,E2 -14589.694} C_VEL
LIN {X 0,Y 333.787,Z 266.524,A -85,B 0,C 180,E1 -14593.39,E2 -14593.39} C_VEL
LIN {X 0,Y 333.736,Z 266.532,A -85,B 0,C 180,E1 -14597.145,E2 -14597.145} C_VEL
LIN {X 0,Y 333.737,Z 266.536,A -85,B 0,C 180,E1 -14599.688,E2 -14599.688} C_VEL
LIN {X 0,Y 333.67,Z 266.541,A -85,B 0,C 180,E1 -14603.588,E2 -14603.588} C_VEL
LIN {X 0,Y 333.725,Z 266.539,A -85,B 0,C 180,E1 -14606.245,E2 -14606.245} C_VEL
LIN {X 0,Y 333.7,Z 266.539,A -85,B 0,C 180,E1 -14608.971,E2 -14608.971} C_VEL
LIN {X 0,Y 333.631,Z 266.549,A -85,B 0,C 180,E1 -14612.586,E2 -14612.586} C_VEL
LIN {X 0,Y 333.665,Z 266.538,A -85,B 0,C 180,E1 -14616.138,E2 -14616.138} C_VEL
LIN {X 0,Y 333.67,Z 266.536,A -85,B 0,C 180,E1 -14619.186,E2 -14619.186} C_VEL
LIN {X 0,Y 333.724,Z 266.664,A -85,B 0,C 180,E1 -14622.213,E2 -14622.213} C_VEL
LIN {X 0,Y 335.786,Z 273.935,A -85,B 0,C 180,E1 -14624.664,E2 -14624.664} C_VEL
LIN {X 0,Y 344.565,Z 290.673,A -85,B 0,C 180,E1 -14626.139,E2 -14626.139} C_VEL
LIN {X 0,Y 351.11,Z 304.508,A -85,B 0,C 180,E1 -14627.201,E2 -14627.201} C_VEL
LIN {X 0,Y 353.516,Z 310.153,A -85,B 0,C 180,E1 -14627.591,E2 -14627.591} C_VEL
LIN {X 0,Y 350.472,Z 409.931,A -85,B 0,C 180,E1 -14629.691,E2 -14629.691} C_VEL
LIN {X 0,Y 349.578,Z 423.856,A -85,B 0,C 180,E1 -14630.195,E2 -14630.195} C_VEL
LIN {X 0,Y 348.285,Z 437.436,A -85,B 0,C 180,E1 -14630.908,E2 -14630.908} C_VEL
LIN {X 0,Y 346.835,Z 450.382,A -85,B 0,C 180,E1 -14631.83,E2 -14631.83} C_VEL
LIN {X 0,Y 344.94,Z 463.783,A -85,B 0,C 180,E1 -14633.056,E2 -14633.056} C_VEL
LIN {X 0,Y 342.963,Z 475.85,A -85,B 0,C 180,E1 -14634.448,E2 -14634.448} C_VEL
LIN {X 0,Y 341.056,Z 486.399,A -85,B 0,C 180,E1 -14635.945,E2 -14635.945} C_VEL
LIN {X 0,Y 339.056,Z 496.563,A -85,B 0,C 180,E1 -14637.702,E2 -14637.702} C_VEL
LIN {X 0,Y 337.254,Z 505.673,A -85,B 0,C 180,E1 -14639.647,E2 -14639.647} C_VEL
LIN {X 0,Y 335.835,Z 512.814,A -85,B 0,C 180,E1 -14641.509,E2 -14641.509} C_VEL
LIN {X 0,Y 334.404,Z 519.89,A -85,B 0,C 180,E1 -14643.811,E2 -14643.811} C_VEL
LIN {X 0,Y 333.525,Z 524.597,A -85,B 0,C 180,E1 -14645.739,E2 -14645.739} C_VEL
LIN {X 0,Y 332.832,Z 528.246,A -85,B 0,C 180,E1 -14647.662,E2 -14647.662} C_VEL
LIN {X 0,Y 332.21,Z 531.738,A -85,B 0,C 180,E1 -14650.216,E2 -14650.216} C_VEL
LIN {X 0,Y 331.915,Z 533.697,A -85,B 0,C 180,E1 -14652.757,E2 -14652.757} C_VEL
LIN {X 0,Y 331.764,Z 534.211,A -85,B 0,C 180,E1 -14655.274,E2 -14655.274} C_VEL
LIN {X 0,Y 331.836,Z 533.335,A -85,B 0,C 180,E1 -14657.773,E2 -14657.773} C_VEL
LIN {X 0,Y 331.903,Z 531.086,A -85,B 0,C 180,E1 -14660.248,E2 -14660.248} C_VEL
LIN {X 0,Y 332.286,Z 527.412,A -85,B 0,C 180,E1 -14662.71,E2 -14662.71} C_VEL
LIN {X 0,Y 332.64,Z 523.668,A -85,B 0,C 180,E1 -14664.545,E2 -14664.545} C_VEL
LIN {X 0,Y 333.08,Z 519.034,A -85,B 0,C 180,E1 -14666.371,E2 -14666.371} C_VEL
LIN {X 0,Y 333.798,Z 512.297,A -85,B 0,C 180,E1 -14668.492,E2 -14668.492} C_VEL
LIN {X 0,Y 334.756,Z 505.247,A -85,B 0,C 180,E1 -14670.301,E2 -14670.301} C_VEL
LIN {X 0,Y 335.95,Z 496.778,A -85,B 0,C 180,E1 -14672.098,E2 -14672.098} C_VEL
LIN {X 0,Y 337.317,Z 486.56,A -85,B 0,C 180,E1 -14673.883,E2 -14673.883} C_VEL
LIN {X 0,Y 338.844,Z 475.229,A -85,B 0,C 180,E1 -14675.49,E2 -14675.49} C_VEL
LIN {X 0,Y 340.243,Z 463.252,A -85,B 0,C 180,E1 -14676.873,E2 -14676.873} C_VEL
LIN {X 0,Y 341.509,Z 451.307,A -85,B 0,C 180,E1 -14677.985,E2 -14677.985} C_VEL
LIN {X 0,Y 342.679,Z 437.442,A -85,B 0,C 180,E1 -14678.997,E2 -14678.997} C_VEL
LIN {X 0,Y 343.628,Z 423.432,A -85,B 0,C 180,E1 -14679.751,E2 -14679.751} C_VEL
LIN {X 0,Y 344.243,Z 409.844,A -85,B 0,C 180,E1 -14680.253,E2 -14680.253} C_VEL
LIN {X 0,Y 346.755,Z 307.066,A -85,B 0,C 180,E1 -14682.401,E2 -14682.401} C_VEL
LIN {X 0,Y 344.881,Z 298.325,A -85,B 0,C 180,E1 -14682.726,E2 -14682.726} C_VEL
LIN {X 0,Y 337.302,Z 278.239,A -85,B 0,C 180,E1 -14683.73,E2 -14683.73} C_VEL
LIN {X 0,Y 335.634,Z 275.239,A -85,B 0,C 180,E1 -14684.005,E2 -14684.005} C_VEL
LIN {X 0,Y 333.386,Z 272.322,A -85,B 0,C 180,E1 -14684.529,E2 -14684.529} C_VEL
LIN {X 0,Y 331.214,Z 270.22,A -85,B 0,C 180,E1 -14685.185,E2 -14685.185} C_VEL
LIN {X 0,Y 328.935,Z 268.579,A -85,B 0,C 180,E1 -14686.109,E2 -14686.109} C_VEL
LIN {X 0,Y 327.298,Z 267.69,A -85,B 0,C 180,E1 -14687.123,E2 -14687.123} C_VEL
LIN {X 0,Y 326.689,Z 267.415,A -85,B 0,C 180,E1 -14688.183,E2 -14688.183} C_VEL
LIN {X 0,Y 326.64,Z 267.423,A -85,B 0,C 180,E1 -14691.455,E2 -14691.455} C_VEL
LIN {X 0,Y 326.677,Z 267.418,A -85,B 0,C 180,E1 -14695.484,E2 -14695.484} C_VEL
LIN {X 0,Y 326.648,Z 267.421,A -85,B 0,C 180,E1 -14699.66,E2 -14699.66} C_VEL
LIN {X 0,Y 326.594,Z 267.427,A -85,B 0,C 180,E1 -14704.02,E2 -14704.02} C_VEL
LIN {X 0,Y 326.618,Z 267.425,A -85,B 0,C 180,E1 -14707.24,E2 -14707.24} C_VEL
LIN {X 0,Y 326.623,Z 267.419,A -85,B 0,C 180,E1 -14710.203,E2 -14710.203} C_VEL
LIN {X 0,Y 326.646,Z 267.422,A -85,B 0,C 180,E1 -14713.511,E2 -14713.511} C_VEL
LIN {X 0,Y 326.638,Z 267.42,A -85,B 0,C 180,E1 -14717.015,E2 -14717.015} C_VEL
LIN {X 0,Y 326.633,Z 267.422,A -85,B 0,C 180,E1 -14720.767,E2 -14720.767} C_VEL
LIN {X 0,Y 326.601,Z 267.42,A -85,B 0,C 180,E1 -14724.482,E2 -14724.482} C_VEL
LIN {X 0,Y 326.597,Z 267.427,A -85,B 0,C 180,E1 -14727.457,E2 -14727.457} C_VEL
LIN {X 0,Y 326.65,Z 267.418,A -85,B 0,C 180,E1 -14730.342,E2 -14730.342} C_VEL
LIN {X 0,Y 326.68,Z 267.412,A -85,B 0,C 180,E1 -14734.518,E2 -14734.518} C_VEL
LIN {X 0,Y 326.639,Z 267.422,A -85,B 0,C 180,E1 -14738.547,E2 -14738.547} C_VEL
LIN {X 0,Y 326.736,Z 267.41,A -85,B 0,C 180,E1 -14741.179,E2 -14741.179} C_VEL
LIN {X 0,Y 326.755,Z 267.404,A -85,B 0,C 180,E1 -14745.435,E2 -14745.435} C_VEL
LIN {X 0,Y 326.761,Z 267.408,A -85,B 0,C 180,E1 -14748.841,E2 -14748.841} C_VEL
LIN {X 0,Y 326.951,Z 267.38,A -85,B 0,C 180,E1 -14752.592,E2 -14752.592} C_VEL
LIN {X 0,Y 326.771,Z 267.403,A -85,B 0,C 180,E1 -14755.066,E2 -14755.066} C_VEL
LIN {X 0,Y 327.042,Z 267.369,A -85,B 0,C 180,E1 -14757.538,E2 -14757.538} C_VEL
LIN {X 0,Y 327.192,Z 267.352,A -85,B 0,C 180,E1 -14760.002,E2 -14760.002} C_VEL
LIN {X 0,Y 327.042,Z 267.369,A -85,B 0,C 180,E1 -14762.465,E2 -14762.465} C_VEL
LIN {X 0,Y 326.984,Z 267.379,A -85,B 0,C 180,E1 -14766.171,E2 -14766.171} C_VEL
LIN {X 0,Y 326.801,Z 267.401,A -85,B 0,C 180,E1 -14769.908,E2 -14769.908} C_VEL
LIN {X 0,Y 326.755,Z 267.402,A -85,B 0,C 180,E1 -14773.687,E2 -14773.687} C_VEL
LIN {X 0,Y 326.696,Z 267.413,A -85,B 0,C 180,E1 -14777.53,E2 -14777.53} C_VEL
LIN {X 0,Y 326.655,Z 267.422,A -85,B 0,C 180,E1 -14780.137,E2 -14780.137} C_VEL
LIN {X 0,Y 326.647,Z 267.423,A -85,B 0,C 180,E1 -14784.131,E2 -14784.131} C_VEL
LIN {X 0,Y 326.683,Z 267.413,A -85,B 0,C 180,E1 -14786.859,E2 -14786.859} C_VEL
LIN {X 0,Y 326.641,Z 267.419,A -85,B 0,C 180,E1 -14790.613,E2 -14790.613} C_VEL
LIN {X 0,Y 326.608,Z 267.427,A -85,B 0,C 180,E1 -14794.021,E2 -14794.021} C_VEL
LIN {X 0,Y 326.628,Z 267.422,A -85,B 0,C 180,E1 -14797.24,E2 -14797.24} C_VEL
LIN {X 0,Y 326.578,Z 267.428,A -85,B 0,C 180,E1 -14801.133,E2 -14801.133} C_VEL
LIN {X 0,Y 326.528,Z 267.434,A -85,B 0,C 180,E1 -14804.744,E2 -14804.744} C_VEL
LIN {X 0,Y 326.577,Z 267.429,A -85,B 0,C 180,E1 -14808.155,E2 -14808.155} C_VEL
LIN {X 0,Y 326.625,Z 267.426,A -85,B 0,C 180,E1 -14811.392,E2 -14811.392} C_VEL
LIN {X 0,Y 326.64,Z 267.422,A -85,B 0,C 180,E1 -14815.238,E2 -14815.238} C_VEL
LIN {X 0,Y 326.631,Z 267.48,A -85,B 0,C 180,E1 -14815.984,E2 -14815.984} C_VEL
LIN {X 0,Y 329.392,Z 279.478,A -85,B 0,C 180,E1 -14819.199,E2 -14819.199} C_VEL
LIN {X 0,Y 331.543,Z 289.559,A -85,B 0,C 180,E1 -14821.726,E2 -14821.726} C_VEL
LIN {X 0,Y 334.052,Z 296.795,A -85,B 0,C 180,E1 -14822.084,E2 -14822.084} C_VEL
LIN {X 0,Y 339.715,Z 332.212,A -85,B 0,C 180,E1 -14823.306,E2 -14823.306} C_VEL
LIN {X 0,Y 337.495,Z 426.202,A -85,B 0,C 180,E1 -14825.306,E2 -14825.306} C_VEL
LIN {X 0,Y 336.748,Z 440.644,A -85,B 0,C 180,E1 -14825.822,E2 -14825.822} C_VEL
LIN {X 0,Y 335.61,Z 454.476,A -85,B 0,C 180,E1 -14826.555,E2 -14826.555} C_VEL
LIN {X 0,Y 334.397,Z 467.002,A -85,B 0,C 180,E1 -14827.446,E2 -14827.446} C_VEL
LIN {X 0,Y 333.068,Z 479.291,A -85,B 0,C 180,E1 -14828.564,E2 -14828.564} C_VEL
LIN {X 0,Y 331.544,Z 490.759,A -85,B 0,C 180,E1 -14829.851,E2 -14829.851} C_VEL
LIN {X 0,Y 330.073,Z 501.804,A -85,B 0,C 180,E1 -14831.375,E2 -14831.375} C_VEL
LIN {X 0,Y 328.539,Z 512.69,A -85,B 0,C 180,E1 -14833.215,E2 -14833.215} C_VEL
LIN {X 0,Y 327.311,Z 522.382,A -85,B 0,C 180,E1 -14835.233,E2 -14835.233} C_VEL
LIN {X 0,Y 326.397,Z 530.261,A -85,B 0,C 180,E1 -14837.25,E2 -14837.25} C_VEL
LIN {X 0,Y 325.588,Z 537.153,A -85,B 0,C 180,E1 -14839.428,E2 -14839.428} C_VEL
LIN {X 0,Y 325.204,Z 541.883,A -85,B 0,C 180,E1 -14841.299,E2 -14841.299} C_VEL
LIN {X 0,Y 324.963,Z 546.77,A -85,B 0,C 180,E1 -14843.792,E2 -14843.792} C_VEL
LIN {X 0,Y 324.883,Z 550.132,A -85,B 0,C 180,E1 -14846.279,E2 -14846.279} C_VEL
LIN {X 0,Y 324.837,Z 552.063,A -85,B 0,C 180,E1 -14848.76,E2 -14848.76} C_VEL
LIN {X 0,Y 324.875,Z 552.517,A -85,B 0,C 180,E1 -14850,E2 -14850} C_VEL
LIN {X 0,Y 324.829,Z 552.414,A -85,B 0,C 180,E1 -14852.48,E2 -14852.48} C_VEL
LIN {X 0,Y 324.872,Z 550.982,A -85,B 0,C 180,E1 -14854.964,E2 -14854.964} C_VEL
LIN {X 0,Y 325.105,Z 548.2,A -85,B 0,C 180,E1 -14857.452,E2 -14857.452} C_VEL
LIN {X 0,Y 325.604,Z 543.998,A -85,B 0,C 180,E1 -14859.943,E2 -14859.943} C_VEL
LIN {X 0,Y 326.557,Z 538.26,A -85,B 0,C 180,E1 -14862.428,E2 -14862.428} C_VEL
LIN {X 0,Y 327.711,Z 531.825,A -85,B 0,C 180,E1 -14864.595,E2 -14864.595} C_VEL
LIN {X 0,Y 329.265,Z 523.866,A -85,B 0,C 180,E1 -14866.747,E2 -14866.747} C_VEL
LIN {X 0,Y 331.016,Z 515.567,A -85,B 0,C 180,E1 -14868.57,E2 -14868.57} C_VEL
LIN {X 0,Y 333.103,Z 505.613,A -85,B 0,C 180,E1 -14870.372,E2 -14870.372} C_VEL
LIN {X 0,Y 335.268,Z 494.568,A -85,B 0,C 180,E1 -14872.005,E2 -14872.005} C_VEL
LIN {X 0,Y 337.385,Z 482.289,A -85,B 0,C 180,E1 -14873.471,E2 -14873.471} C_VEL
LIN {X 0,Y 339.355,Z 470.067,A -85,B 0,C 180,E1 -14874.631,E2 -14874.631} C_VEL
LIN {X 0,Y 341.183,Z 456.563,A -85,B 0,C 180,E1 -14875.63,E2 -14875.63} C_VEL
LIN {X 0,Y 342.747,Z 442.413,A -85,B 0,C 180,E1 -14876.403,E2 -14876.403} C_VEL
LIN {X 0,Y 343.86,Z 428.489,A -85,B 0,C 180,E1 -14876.925,E2 -14876.925} C_VEL
LIN {X 0,Y 344.905,Z 399.545,A -85,B 0,C 180,E1 -14877.576,E2 -14877.576} C_VEL
LIN {X 0,Y 346.842,Z 333.805,A -85,B 0,C 180,E1 -14878.974,E2 -14878.974} C_VEL
LIN {X 0,Y 342.162,Z 309.762,A -85,B 0,C 180,E1 -14880.087,E2 -14880.087} C_VEL
LIN {X 0,Y 338.195,Z 300.696,A -85,B 0,C 180,E1 -14880.78,E2 -14880.78} C_VEL
LIN {X 0,Y 332.205,Z 288.294,A -85,B 0,C 180,E1 -14881.879,E2 -14881.879} C_VEL
LIN {X 0,Y 329.526,Z 277.604,A -85,B 0,C 180,E1 -14885.158,E2 -14885.158} C_VEL
LIN {X 0,Y 326.652,Z 267.424,A -85,B 0,C 180,E1 -14888.603,E2 -14888.603} C_VEL
LIN {X 0,Y 326.622,Z 267.421,A -85,B 0,C 180,E1 -14891.837,E2 -14891.837} C_VEL
LIN {X 0,Y 326.581,Z 267.428,A -85,B 0,C 180,E1 -14895.246,E2 -14895.246} C_VEL
LIN {X 0,Y 326.577,Z 267.431,A -85,B 0,C 180,E1 -14898.867,E2 -14898.867} C_VEL
LIN {X 0,Y 326.626,Z 267.414,A -85,B 0,C 180,E1 -14902.76,E2 -14902.76} C_VEL
LIN {X 0,Y 326.605,Z 267.415,A -85,B 0,C 180,E1 -14905.979,E2 -14905.979} C_VEL
LIN {X 0,Y 326.658,Z 267.421,A -85,B 0,C 180,E1 -14910.339,E2 -14910.339} C_VEL
LIN {X 0,Y 326.687,Z 267.415,A -85,B 0,C 180,E1 -14914.515,E2 -14914.515} C_VEL
LIN {X 0,Y 326.642,Z 267.42,A -85,B 0,C 180,E1 -14918.544,E2 -14918.544} C_VEL
LIN {X 0,Y 326.74,Z 267.406,A -85,B 0,C 180,E1 -14921.176,E2 -14921.176} C_VEL
LIN {X 0,Y 326.758,Z 267.405,A -85,B 0,C 180,E1 -14925.432,E2 -14925.432} C_VEL
LIN {X 0,Y 326.764,Z 267.398,A -85,B 0,C 180,E1 -14928.837,E2 -14928.837} C_VEL
LIN {X 0,Y 326.96,Z 267.371,A -85,B 0,C 180,E1 -14932.588,E2 -14932.588} C_VEL
LIN {X 0,Y 326.771,Z 267.408,A -85,B 0,C 180,E1 -14935.063,E2 -14935.063} C_VEL
LIN {X 0,Y 327.04,Z 267.365,A -85,B 0,C 180,E1 -14937.535,E2 -14937.535} C_VEL
LIN {X 0,Y 327.21,Z 267.348,A -85,B 0,C 180,E1 -14939.998,E2 -14939.998} C_VEL
LIN {X 0,Y 327.04,Z 267.368,A -85,B 0,C 180,E1 -14942.462,E2 -14942.462} C_VEL
LIN {X 0,Y 326.953,Z 267.377,A -85,B 0,C 180,E1 -14946.667,E2 -14946.667} C_VEL
LIN {X 0,Y 326.803,Z 267.393,A -85,B 0,C 180,E1 -14949.905,E2 -14949.905} C_VEL
LIN {X 0,Y 326.749,Z 267.4,A -85,B 0,C 180,E1 -14953.684,E2 -14953.684} C_VEL
LIN {X 0,Y 326.689,Z 267.41,A -85,B 0,C 180,E1 -14957.526,E2 -14957.526} C_VEL
LIN {X 0,Y 326.663,Z 267.416,A -85,B 0,C 180,E1 -14960.133,E2 -14960.133} C_VEL
LIN {X 0,Y 326.647,Z 267.415,A -85,B 0,C 180,E1 -14964.127,E2 -14964.127} C_VEL
LIN {X 0,Y 326.674,Z 267.414,A -85,B 0,C 180,E1 -14966.856,E2 -14966.856} C_VEL
LIN {X 0,Y 326.627,Z 267.405,A -85,B 0,C 180,E1 -14970.61,E2 -14970.61} C_VEL
LIN {X 0,Y 326.594,Z 267.421,A -85,B 0,C 180,E1 -14974.018,E2 -14974.018} C_VEL
LIN {X 0,Y 326.617,Z 267.428,A -85,B 0,C 180,E1 -14977.238,E2 -14977.238} C_VEL
LIN {X 0,Y 326.662,Z 267.416,A -85,B 0,C 180,E1 -14981.307,E2 -14981.307} C_VEL
LIN {X 0,Y 328.493,Z 273.995,A -85,B 0,C 180,E1 -14983.731,E2 -14983.731} C_VEL
LIN {X 0,Y 330.625,Z 277.914,A -85,B 0,C 180,E1 -14984.116,E2 -14984.116} C_VEL
LIN {X 0,Y 338.813,Z 293.25,A -85,B 0,C 180,E1 -14985.533,E2 -14985.533} C_VEL
LIN {X 0,Y 346.235,Z 309.166,A -85,B 0,C 180,E1 -14986.786,E2 -14986.786} C_VEL
LIN {X 0,Y 347.542,Z 312.389,A -85,B 0,C 180,E1 -14987.008,E2 -14987.008} C_VEL
LIN {X 0,Y 344.381,Z 410.273,A -85,B 0,C 180,E1 -14989.097,E2 -14989.097} C_VEL
LIN {X 0,Y 343.415,Z 424.461,A -85,B 0,C 180,E1 -14989.622,E2 -14989.622} C_VEL
LIN {X 0,Y 342.064,Z 437.929,A -85,B 0,C 180,E1 -14990.343,E2 -14990.343} C_VEL
LIN {X 0,Y 340.433,Z 451.737,A -85,B 0,C 180,E1 -14991.356,E2 -14991.356} C_VEL
LIN {X 0,Y 338.636,Z 463.89,A -85,B 0,C 180,E1 -14992.496,E2 -14992.496} C_VEL
LIN {X 0,Y 336.571,Z 475.563,A -85,B 0,C 180,E1 -14993.852,E2 -14993.852} C_VEL
LIN {X 0,Y 334.525,Z 486.611,A -85,B 0,C 180,E1 -14995.443,E2 -14995.443} C_VEL
LIN {X 0,Y 332.654,Z 495.758,A -85,B 0,C 180,E1 -14997.044,E2 -14997.044} C_VEL
LIN {X 0,Y 330.748,Z 504.898,A -85,B 0,C 180,E1 -14998.985,E2 -14998.985} C_VEL
LIN {X 0,Y 329.031,Z 513.069,A -85,B 0,C 180,E1 -15001.129,E2 -15001.129} C_VEL
LIN {X 0,Y 327.666,Z 519.487,A -85,B 0,C 180,E1 -15003.23,E2 -15003.23} C_VEL
LIN {X 0,Y 326.67,Z 524.277,A -85,B 0,C 180,E1 -15005.196,E2 -15005.196} C_VEL
LIN {X 0,Y 325.889,Z 528.058,A -85,B 0,C 180,E1 -15007.159,E2 -15007.159} C_VEL
LIN {X 0,Y 325.542,Z 530.064,A -85,B 0,C 180,E1 -15008.47,E2 -15008.47} C_VEL
LIN {X 0,Y 324.983,Z 532.912,A -85,B 0,C 180,E1 -15011.072,E2 -15011.072} C_VEL
LIN {X 0,Y 324.874,Z 533.781,A -85,B 0,C 180,E1 -15012.371,E2 -15012.371} C_VEL
LIN {X 0,Y 324.661,Z 534.442,A -85,B 0,C 180,E1 -15014.944,E2 -15014.944} C_VEL
LIN {X 0,Y 324.759,Z 533.68,A -85,B 0,C 180,E1 -15017.502,E2 -15017.502} C_VEL
LIN {X 0,Y 324.784,Z 531.547,A -85,B 0,C 180,E1 -15020.032,E2 -15020.032} C_VEL
LIN {X 0,Y 325.166,Z 527.99,A -85,B 0,C 180,E1 -15022.549,E2 -15022.549} C_VEL
LIN {X 0,Y 325.62,Z 522.942,A -85,B 0,C 180,E1 -15025.048,E2 -15025.048} C_VEL
LIN {X 0,Y 326.173,Z 518.057,A -85,B 0,C 180,E1 -15026.912,E2 -15026.912} C_VEL
LIN {X 0,Y 326.978,Z 511.045,A -85,B 0,C 180,E1 -15029.076,E2 -15029.076} C_VEL
LIN {X 0,Y 328.199,Z 502.356,A -85,B 0,C 180,E1 -15031.227,E2 -15031.227} C_VEL
LIN {X 0,Y 329.513,Z 493.272,A -85,B 0,C 180,E1 -15033.057,E2 -15033.057} C_VEL
LIN {X 0,Y 331.063,Z 482.279,A -85,B 0,C 180,E1 -15034.871,E2 -15034.871} C_VEL
LIN {X 0,Y 332.591,Z 470.88,A -85,B 0,C 180,E1 -15036.391,E2 -15036.391} C_VEL
LIN {X 0,Y 333.946,Z 458.723,A -85,B 0,C 180,E1 -15037.71,E2 -15037.71} C_VEL
LIN {X 0,Y 335.264,Z 446.79,A -85,B 0,C 180,E1 -15038.742,E2 -15038.742} C_VEL
LIN {X 0,Y 336.302,Z 433.821,A -85,B 0,C 180,E1 -15039.624,E2 -15039.624} C_VEL
LIN {X 0,Y 337.153,Z 419.878,A -85,B 0,C 180,E1 -15040.319,E2 -15040.319} C_VEL
LIN {X 0,Y 337.756,Z 405.27,A -85,B 0,C 180,E1 -15040.793,E2 -15040.793} C_VEL
LIN {X 0,Y 340.182,Z 307.419,A -85,B 0,C 180,E1 -15042.853,E2 -15042.853} C_VEL
LIN {X 0,Y 338.425,Z 300.16,A -85,B 0,C 180,E1 -15043.145,E2 -15043.145} C_VEL
LIN {X 0,Y 329.21,Z 276.105,A -85,B 0,C 180,E1 -15044.401,E2 -15044.401} C_VEL
LIN {X 0,Y 327.986,Z 273.133,A -85,B 0,C 180,E1 -15044.571,E2 -15044.571} C_VEL
LIN {X 0,Y 326.708,Z 267.415,A -85,B 0,C 180,E1 -15046.319,E2 -15046.319} C_VEL
LIN {X 0,Y 326.689,Z 267.415,A -85,B 0,C 180,E1 -15048.183,E2 -15048.183} C_VEL
LIN {X 0,Y 326.044,Z 267.498,A -85,B 0,C 180,E1 -15049.211,E2 -15049.211} C_VEL
LIN {X 0,Y 323.161,Z 267.857,A -85,B 0,C 180,E1 -15050.884,E2 -15050.884} C_VEL
LIN {X 0,Y 320.696,Z 268.165,A -85,B 0,C 180,E1 -15052.239,E2 -15052.239} C_VEL
LIN {X 0,Y 319.636,Z 268.295,A -85,B 0,C 180,E1 -15053.289,E2 -15053.289} C_VEL
LIN {X 0,Y 319.55,Z 268.303,A -85,B 0,C 180,E1 -15053.645,E2 -15053.645} C_VEL
LIN {X 0,Y 319.622,Z 268.295,A -85,B 0,C 180,E1 -15056.089,E2 -15056.089} C_VEL
LIN {X 0,Y 319.577,Z 268.299,A -85,B 0,C 180,E1 -15058.934,E2 -15058.934} C_VEL
LIN {X 0,Y 319.52,Z 268.309,A -85,B 0,C 180,E1 -15061.863,E2 -15061.863} C_VEL
LIN {X 0,Y 319.568,Z 268.304,A -85,B 0,C 180,E1 -15065.544,E2 -15065.544} C_VEL
LIN {X 0,Y 319.588,Z 268.299,A -85,B 0,C 180,E1 -15068.005,E2 -15068.005} C_VEL
LIN {X 0,Y 319.59,Z 268.301,A -85,B 0,C 180,E1 -15071.613,E2 -15071.613} C_VEL
LIN {X 0,Y 319.633,Z 268.295,A -85,B 0,C 180,E1 -15075.286,E2 -15075.286} C_VEL
LIN {X 0,Y 319.571,Z 268.299,A -85,B 0,C 180,E1 -15078.721,E2 -15078.721} C_VEL
LIN {X 0,Y 319.571,Z 268.298,A -85,B 0,C 180,E1 -15082.344,E2 -15082.344} C_VEL
LIN {X 0,Y 319.549,Z 268.302,A -85,B 0,C 180,E1 -15085.125,E2 -15085.125} C_VEL
LIN {X 0,Y 319.56,Z 268.306,A -85,B 0,C 180,E1 -15089.059,E2 -15089.059} C_VEL
LIN {X 0,Y 319.599,Z 268.293,A -85,B 0,C 180,E1 -15092.5,E2 -15092.5} C_VEL
LIN {X 0,Y 319.595,Z 268.298,A -85,B 0,C 180,E1 -15095.305,E2 -15095.305} C_VEL
LIN {X 0,Y 319.588,Z 268.298,A -85,B 0,C 180,E1 -15098.049,E2 -15098.049} C_VEL
LIN {X 0,Y 319.68,Z 268.29,A -85,B 0,C 180,E1 -15100.964,E2 -15100.964} C_VEL
LIN {X 0,Y 319.723,Z 268.281,A -85,B 0,C 180,E1 -15105.278,E2 -15105.278} C_VEL
LIN {X 0,Y 319.745,Z 268.278,A -85,B 0,C 180,E1 -15109.874,E2 -15109.874} C_VEL
LIN {X 0,Y 319.906,Z 268.257,A -85,B 0,C 180,E1 -15112.427,E2 -15112.427} C_VEL
LIN {X 0,Y 319.74,Z 268.279,A -85,B 0,C 180,E1 -15114.958,E2 -15114.958} C_VEL
LIN {X 0,Y 319.985,Z 268.248,A -85,B 0,C 180,E1 -15117.484,E2 -15117.484} C_VEL
LIN {X 0,Y 320.144,Z 268.229,A -85,B 0,C 180,E1 -15120.002,E2 -15120.002} C_VEL
LIN {X 0,Y 319.985,Z 268.246,A -85,B 0,C 180,E1 -15122.519,E2 -15122.519} C_VEL
LIN {X 0,Y 319.939,Z 268.257,A -85,B 0,C 180,E1 -15126.307,E2 -15126.307} C_VEL
LIN {X 0,Y 319.833,Z 268.268,A -85,B 0,C 180,E1 -15128.85,E2 -15128.85} C_VEL
LIN {X 0,Y 319.677,Z 268.284,A -85,B 0,C 180,E1 -15132.702,E2 -15132.702} C_VEL
LIN {X 0,Y 319.696,Z 268.283,A -85,B 0,C 180,E1 -15135.297,E2 -15135.297} C_VEL
LIN {X 0,Y 319.649,Z 268.289,A -85,B 0,C 180,E1 -15139.258,E2 -15139.258} C_VEL
LIN {X 0,Y 319.558,Z 268.301,A -85,B 0,C 180,E1 -15143.322,E2 -15143.322} C_VEL
LIN {X 0,Y 319.633,Z 268.296,A -85,B 0,C 180,E1 -15146.09,E2 -15146.09} C_VEL
LIN {X 0,Y 319.589,Z 268.298,A -85,B 0,C 180,E1 -15148.935,E2 -15148.935} C_VEL
LIN {X 0,Y 319.538,Z 268.308,A -85,B 0,C 180,E1 -15151.863,E2 -15151.863} C_VEL
LIN {X 0,Y 319.58,Z 268.301,A -85,B 0,C 180,E1 -15155.544,E2 -15155.544} C_VEL
LIN {X 0,Y 319.573,Z 268.304,A -85,B 0,C 180,E1 -15158.01,E2 -15158.01} C_VEL
LIN {X 0,Y 319.526,Z 268.31,A -85,B 0,C 180,E1 -15161.598,E2 -15161.598} C_VEL
LIN {X 0,Y 319.489,Z 268.313,A -85,B 0,C 180,E1 -15165.258,E2 -15165.258} C_VEL
LIN {X 0,Y 319.53,Z 268.306,A -85,B 0,C 180,E1 -15168.713,E2 -15168.713} C_VEL
LIN {X 0,Y 319.563,Z 268.303,A -85,B 0,C 180,E1 -15172.349,E2 -15172.349} C_VEL
LIN {X 0,Y 319.604,Z 268.376,A -85,B 0,C 180,E1 -15175.549,E2 -15175.549} C_VEL
LIN {X 0,Y 322.315,Z 280.238,A -85,B 0,C 180,E1 -15178.812,E2 -15178.812} C_VEL
LIN {X 0,Y 324.161,Z 289.086,A -85,B 0,C 180,E1 -15181.137,E2 -15181.137} C_VEL
LIN {X 0,Y 327.748,Z 299.013,A -85,B 0,C 180,E1 -15181.657,E2 -15181.657} C_VEL
LIN {X 0,Y 333.132,Z 333.471,A -85,B 0,C 180,E1 -15182.868,E2 -15182.868} C_VEL
LIN {X 0,Y 330.875,Z 425.604,A -85,B 0,C 180,E1 -15184.862,E2 -15184.862} C_VEL
LIN {X 0,Y 330.132,Z 440.251,A -85,B 0,C 180,E1 -15185.389,E2 -15185.389} C_VEL
LIN {X 0,Y 328.918,Z 454.135,A -85,B 0,C 180,E1 -15186.132,E2 -15186.132} C_VEL
LIN {X 0,Y 327.579,Z 467.589,A -85,B 0,C 180,E1 -15187.117,E2 -15187.117} C_VEL
LIN {X 0,Y 326.048,Z 480.909,A -85,B 0,C 180,E1 -15188.382,E2 -15188.382} C_VEL
LIN {X 0,Y 324.527,Z 492.28,A -85,B 0,C 180,E1 -15189.727,E2 -15189.727} C_VEL
LIN {X 0,Y 322.987,Z 503.029,A -85,B 0,C 180,E1 -15191.28,E2 -15191.28} C_VEL
LIN {X 0,Y 321.447,Z 513.682,A -85,B 0,C 180,E1 -15193.161,E2 -15193.161} C_VEL
LIN {X 0,Y 320.267,Z 522.558,A -85,B 0,C 180,E1 -15195.081,E2 -15195.081} C_VEL
LIN {X 0,Y 319.284,Z 530.86,A -85,B 0,C 180,E1 -15197.284,E2 -15197.284} C_VEL
LIN {X 0,Y 318.555,Z 536.698,A -85,B 0,C 180,E1 -15199.192,E2 -15199.192} C_VEL
LIN {X 0,Y 318.141,Z 541.483,A -85,B 0,C 180,E1 -15201.104,E2 -15201.104} C_VEL
LIN {X 0,Y 317.892,Z 546.422,A -85,B 0,C 180,E1 -15203.654,E2 -15203.654} C_VEL
LIN {X 0,Y 317.79,Z 549.832,A -85,B 0,C 180,E1 -15206.196,E2 -15206.196} C_VEL
LIN {X 0,Y 317.748,Z 551.82,A -85,B 0,C 180,E1 -15208.732,E2 -15208.732} C_VEL
LIN {X 0,Y 317.783,Z 552.3,A -85,B 0,C 180,E1 -15210,E2 -15210} C_VEL
LIN {X 0,Y 317.75,Z 552.246,A -85,B 0,C 180,E1 -15212.535,E2 -15212.535} C_VEL
LIN {X 0,Y 317.789,Z 550.859,A -85,B 0,C 180,E1 -15215.075,E2 -15215.075} C_VEL
LIN {X 0,Y 318.027,Z 548.122,A -85,B 0,C 180,E1 -15217.619,E2 -15217.619} C_VEL
LIN {X 0,Y 318.564,Z 543.968,A -85,B 0,C 180,E1 -15220.165,E2 -15220.165} C_VEL
LIN {X 0,Y 319.613,Z 538.281,A -85,B 0,C 180,E1 -15222.702,E2 -15222.702} C_VEL
LIN {X 0,Y 320.808,Z 531.909,A -85,B 0,C 180,E1 -15224.916,E2 -15224.916} C_VEL
LIN {X 0,Y 322.464,Z 524.02,A -85,B 0,C 180,E1 -15227.111,E2 -15227.111} C_VEL
LIN {X 0,Y 324.291,Z 515.801,A -85,B 0,C 180,E1 -15228.97,E2 -15228.97} C_VEL
LIN {X 0,Y 326.468,Z 505.934,A -85,B 0,C 180,E1 -15230.805,E2 -15230.805} C_VEL
LIN {X 0,Y 328.72,Z 494.999,A -85,B 0,C 180,E1 -15232.467,E2 -15232.467} C_VEL
LIN {X 0,Y 330.995,Z 482.45,A -85,B 0,C 180,E1 -15234.008,E2 -15234.008} C_VEL
LIN {X 0,Y 332.962,Z 470.896,A -85,B 0,C 180,E1 -15235.137,E2 -15235.137} C_VEL
LIN {X 0,Y 334.857,Z 457.676,A -85,B 0,C 180,E1 -15236.151,E2 -15236.151} C_VEL
LIN {X 0,Y 336.499,Z 443.974,A -85,B 0,C 180,E1 -15236.933,E2 -15236.933} C_VEL
LIN {X 0,Y 337.713,Z 429.797,A -85,B 0,C 180,E1 -15237.498,E2 -15237.498} C_VEL
LIN {X 0,Y 338.609,Z 409.467,A -85,B 0,C 180,E1 -15237.986,E2 -15237.986} C_VEL
LIN {X 0,Y 340.879,Z 334.853,A -85,B 0,C 180,E1 -15239.602,E2 -15239.602} C_VEL
LIN {X 0,Y 336.435,Z 311.945,A -85,B 0,C 180,E1 -15240.7,E2 -15240.7} C_VEL
LIN {X 0,Y 328.932,Z 296.093,A -85,B 0,C 180,E1 -15242.043,E2 -15242.043} C_VEL
LIN {X 0,Y 324.959,Z 288.187,A -85,B 0,C 180,E1 -15242.793,E2 -15242.793} C_VEL
LIN {X 0,Y 322.302,Z 277.923,A -85,B 0,C 180,E1 -15246.067,E2 -15246.067} C_VEL
LIN {X 0,Y 319.599,Z 268.302,A -85,B 0,C 180,E1 -15249.416,E2 -15249.416} C_VEL
LIN {X 0,Y 319.597,Z 268.299,A -85,B 0,C 180,E1 -15253.473,E2 -15253.473} C_VEL
LIN {X 0,Y 319.564,Z 268.304,A -85,B 0,C 180,E1 -15257.017,E2 -15257.017} C_VEL
LIN {X 0,Y 319.546,Z 268.303,A -85,B 0,C 180,E1 -15260.369,E2 -15260.369} C_VEL
LIN {X 0,Y 319.557,Z 268.281,A -85,B 0,C 180,E1 -15263.571,E2 -15263.571} C_VEL
LIN {X 0,Y 319.575,Z 268.301,A -85,B 0,C 180,E1 -15266.685,E2 -15266.685} C_VEL
LIN {X 0,Y 319.589,Z 268.294,A -85,B 0,C 180,E1 -15269.615,E2 -15269.615} C_VEL
LIN {X 0,Y 319.606,Z 268.291,A -85,B 0,C 180,E1 -15272.496,E2 -15272.496} C_VEL
LIN {X 0,Y 319.601,Z 268.295,A -85,B 0,C 180,E1 -15275.302,E2 -15275.302} C_VEL
LIN {X 0,Y 319.593,Z 268.301,A -85,B 0,C 180,E1 -15278.046,E2 -15278.046} C_VEL
LIN {X 0,Y 319.685,Z 268.284,A -85,B 0,C 180,E1 -15280.961,E2 -15280.961} C_VEL
LIN {X 0,Y 319.726,Z 268.28,A -85,B 0,C 180,E1 -15285.274,E2 -15285.274} C_VEL
LIN {X 0,Y 319.751,Z 268.281,A -85,B 0,C 180,E1 -15289.871,E2 -15289.871} C_VEL
LIN {X 0,Y 319.919,Z 268.248,A -85,B 0,C 180,E1 -15292.424,E2 -15292.424} C_VEL
LIN {X 0,Y 319.74,Z 268.283,A -85,B 0,C 180,E1 -15294.954,E2 -15294.954} C_VEL
LIN {X 0,Y 319.984,Z 268.243,A -85,B 0,C 180,E1 -15297.481,E2 -15297.481} C_VEL
LIN {X 0,Y 320.162,Z 268.226,A -85,B 0,C 180,E1 -15299.998,E2 -15299.998} C_VEL
LIN {X 0,Y 319.983,Z 268.247,A -85,B 0,C 180,E1 -15302.516,E2 -15302.516} C_VEL
LIN {X 0,Y 319.915,Z 268.253,A -85,B 0,C 180,E1 -15306.657,E2 -15306.657} C_VEL
LIN {X 0,Y 319.833,Z 268.266,A -85,B 0,C 180,E1 -15308.846,E2 -15308.846} C_VEL
LIN {X 0,Y 319.672,Z 268.287,A -85,B 0,C 180,E1 -15312.698,E2 -15312.698} C_VEL
LIN {X 0,Y 319.69,Z 268.29,A -85,B 0,C 180,E1 -15315.294,E2 -15315.294} C_VEL
LIN {X 0,Y 319.667,Z 268.291,A -85,B 0,C 180,E1 -15319.253,E2 -15319.253} C_VEL
LIN {X 0,Y 319.563,Z 268.299,A -85,B 0,C 180,E1 -15323.318,E2 -15323.318} C_VEL
LIN {X 0,Y 319.625,Z 268.296,A -85,B 0,C 180,E1 -15326.087,E2 -15326.087} C_VEL
LIN {X 0,Y 319.578,Z 268.299,A -85,B 0,C 180,E1 -15328.932,E2 -15328.932} C_VEL
LIN {X 0,Y 319.52,Z 268.296,A -85,B 0,C 180,E1 -15331.861,E2 -15331.861} C_VEL
LIN {X 0,Y 319.567,Z 268.288,A -85,B 0,C 180,E1 -15335.542,E2 -15335.542} C_VEL
LIN {X 0,Y 319.571,Z 268.298,A -85,B 0,C 180,E1 -15338.006,E2 -15338.006} C_VEL
LIN {X 0,Y 319.58,Z 268.305,A -85,B 0,C 180,E1 -15340.547,E2 -15340.547} C_VEL
LIN {X 0,Y 321.274,Z 274.375,A -85,B 0,C 180,E1 -15342.759,E2 -15342.759} C_VEL
LIN {X 0,Y 328.991,Z 288.126,A -85,B 0,C 180,E1 -15344.179,E2 -15344.179} C_VEL
LIN {X 0,Y 335.458,Z 300.79,A -85,B 0,C 180,E1 -15345.324,E2 -15345.324} C_VEL
LIN {X 0,Y 341.561,Z 314.303,A -85,B 0,C 180,E1 -15346.388,E2 -15346.388} C_VEL
LIN {X 0,Y 338.337,Z 410.619,A -85,B 0,C 180,E1 -15348.483,E2 -15348.483} C_VEL
LIN {X 0,Y 337.344,Z 424.514,A -85,B 0,C 180,E1 -15349.002,E2 -15349.002} C_VEL
LIN {X 0,Y 335.9,Z 438.435,A -85,B 0,C 180,E1 -15349.761,E2 -15349.761} C_VEL
LIN {X 0,Y 334.332,Z 451.241,A -85,B 0,C 180,E1 -15350.71,E2 -15350.71} C_VEL
LIN {X 0,Y 332.392,Z 463.862,A -85,B 0,C 180,E1 -15351.902,E2 -15351.902} C_VEL
LIN {X 0,Y 330.303,Z 475.301,A -85,B 0,C 180,E1 -15353.244,E2 -15353.244} C_VEL
LIN {X 0,Y 328.123,Z 486.42,A -85,B 0,C 180,E1 -15354.857,E2 -15354.857} C_VEL
LIN {X 0,Y 325.973,Z 496.487,A -85,B 0,C 180,E1 -15356.649,E2 -15356.649} C_VEL
LIN {X 0,Y 323.988,Z 505.538,A -85,B 0,C 180,E1 -15358.628,E2 -15358.628} C_VEL
LIN {X 0,Y 322.233,Z 513.349,A -85,B 0,C 180,E1 -15360.735,E2 -15360.735} C_VEL
LIN {X 0,Y 320.929,Z 519.032,A -85,B 0,C 180,E1 -15362.622,E2 -15362.622} C_VEL
LIN {X 0,Y 319.796,Z 524.21,A -85,B 0,C 180,E1 -15364.745,E2 -15364.745} C_VEL
LIN {X 0,Y 318.998,Z 527.869,A -85,B 0,C 180,E1 -15366.637,E2 -15366.637} C_VEL
LIN {X 0,Y 318.225,Z 531.615,A -85,B 0,C 180,E1 -15369.308,E2 -15369.308} C_VEL
LIN {X 0,Y 317.804,Z 533.84,A -85,B 0,C 180,E1 -15371.965,E2 -15371.965} C_VEL
LIN {X 0,Y 317.572,Z 534.629,A -85,B 0,C 180,E1 -15374.6,E2 -15374.6} C_VEL
LIN {X 0,Y 317.661,Z 534.016,A -85,B 0,C 180,E1 -15377.218,E2 -15377.218} C_VEL
LIN {X 0,Y 317.669,Z 532.007,A -85,B 0,C 180,E1 -15379.806,E2 -15379.806} C_VEL
LIN {X 0,Y 318.027,Z 528.569,A -85,B 0,C 180,E1 -15382.381,E2 -15382.381} C_VEL
LIN {X 0,Y 318.405,Z 525.047,A -85,B 0,C 180,E1 -15384.3,E2 -15384.3} C_VEL
LIN {X 0,Y 318.826,Z 520.579,A -85,B 0,C 180,E1 -15386.208,E2 -15386.208} C_VEL
LIN {X 0,Y 319.586,Z 514.139,A -85,B 0,C 180,E1 -15388.425,E2 -15388.425} C_VEL
LIN {X 0,Y 320.718,Z 506.142,A -85,B 0,C 180,E1 -15390.628,E2 -15390.628} C_VEL
LIN {X 0,Y 321.992,Z 497.773,A -85,B 0,C 180,E1 -15392.502,E2 -15392.502} C_VEL
LIN {X 0,Y 323.481,Z 487.709,A -85,B 0,C 180,E1 -15394.361,E2 -15394.361} C_VEL
LIN {X 0,Y 325.089,Z 476.391,A -85,B 0,C 180,E1 -15396.058,E2 -15396.058} C_VEL
LIN {X 0,Y 326.5,Z 465.278,A -85,B 0,C 180,E1 -15397.421,E2 -15397.421} C_VEL
LIN {X 0,Y 327.882,Z 453.103,A -85,B 0,C 180,E1 -15398.629,E2 -15398.629} C_VEL
LIN {X 0,Y 329.192,Z 439.588,A -85,B 0,C 180,E1 -15399.679,E2 -15399.679} C_VEL
LIN {X 0,Y 330.214,Z 425.446,A -85,B 0,C 180,E1 -15400.5,E2 -15400.5} C_VEL
LIN {X 0,Y 330.917,Z 411.527,A -85,B 0,C 180,E1 -15401.058,E2 -15401.058} C_VEL
LIN {X 0,Y 331.753,Z 382.43,A -85,B 0,C 180,E1 -15401.726,E2 -15401.726} C_VEL
LIN {X 0,Y 333.642,Z 309.132,A -85,B 0,C 180,E1 -15403.288,E2 -15403.288} C_VEL
LIN {X 0,Y 332.317,Z 303.041,A -85,B 0,C 180,E1 -15403.528,E2 -15403.528} C_VEL
LIN {X 0,Y 324.249,Z 281.757,A -85,B 0,C 180,E1 -15404.662,E2 -15404.662} C_VEL
LIN {X 0,Y 320.768,Z 273.27,A -85,B 0,C 180,E1 -15405.173,E2 -15405.173} C_VEL
LIN {X 0,Y 319.656,Z 268.294,A -85,B 0,C 180,E1 -15406.69,E2 -15406.69} C_VEL
LIN {X 0,Y 319.664,Z 268.292,A -85,B 0,C 180,E1 -15409.255,E2 -15409.255} C_VEL
LIN {X 0,Y 319.558,Z 268.305,A -85,B 0,C 180,E1 -15413.32,E2 -15413.32} C_VEL
LIN {X 0,Y 319.55,Z 268.303,A -85,B 0,C 180,E1 -15413.645,E2 -15413.645} C_VEL
LIN {X 0,Y 318.884,Z 268.387,A -85,B 0,C 180,E1 -15414.697,E2 -15414.697} C_VEL
LIN {X 0,Y 316.042,Z 268.74,A -85,B 0,C 180,E1 -15416.409,E2 -15416.409} C_VEL
LIN {X 0,Y 313.636,Z 269.042,A -85,B 0,C 180,E1 -15417.797,E2 -15417.797} C_VEL
LIN {X 0,Y 312.608,Z 269.167,A -85,B 0,C 180,E1 -15418.871,E2 -15418.871} C_VEL
LIN {X 0,Y 312.526,Z 269.176,A -85,B 0,C 180,E1 -15419.235,E2 -15419.235} C_VEL
LIN {X 0,Y 312.492,Z 269.182,A -85,B 0,C 180,E1 -15422.667,E2 -15422.667} C_VEL
LIN {X 0,Y 312.524,Z 269.179,A -85,B 0,C 180,E1 -15425.951,E2 -15425.951} C_VEL
LIN {X 0,Y 312.526,Z 269.18,A -85,B 0,C 180,E1 -15429.024,E2 -15429.024} C_VEL
LIN {X 0,Y 312.549,Z 269.174,A -85,B 0,C 180,E1 -15432.421,E2 -15432.421} C_VEL
LIN {X 0,Y 312.581,Z 269.167,A -85,B 0,C 180,E1 -15436.01,E2 -15436.01} C_VEL
LIN {X 0,Y 312.52,Z 269.179,A -85,B 0,C 180,E1 -15439.87,E2 -15439.87} C_VEL
LIN {X 0,Y 312.53,Z 269.176,A -85,B 0,C 180,E1 -15442.618,E2 -15442.618} C_VEL
LIN {X 0,Y 312.509,Z 269.177,A -85,B 0,C 180,E1 -15446.313,E2 -15446.313} C_VEL
LIN {X 0,Y 312.535,Z 269.176,A -85,B 0,C 180,E1 -15450.351,E2 -15450.351} C_VEL
LIN {X 0,Y 312.593,Z 269.163,A -85,B 0,C 180,E1 -15454.066,E2 -15454.066} C_VEL
LIN {X 0,Y 312.578,Z 269.172,A -85,B 0,C 180,E1 -15457.53,E2 -15457.53} C_VEL
LIN {X 0,Y 312.629,Z 269.164,A -85,B 0,C 180,E1 -15461.658,E2 -15461.658} C_VEL
LIN {X 0,Y 312.685,Z 269.156,A -85,B 0,C 180,E1 -15465.688,E2 -15465.688} C_VEL
LIN {X 0,Y 312.691,Z 269.156,A -85,B 0,C 180,E1 -15469.643,E2 -15469.643} C_VEL
LIN {X 0,Y 312.846,Z 269.135,A -85,B 0,C 180,E1 -15472.255,E2 -15472.255} C_VEL
LIN {X 0,Y 312.71,Z 269.155,A -85,B 0,C 180,E1 -15474.844,E2 -15474.844} C_VEL
LIN {X 0,Y 312.984,Z 269.123,A -85,B 0,C 180,E1 -15478.715,E2 -15478.715} C_VEL
LIN {X 0,Y 312.985,Z 269.116,A -85,B 0,C 180,E1 -15481.288,E2 -15481.288} C_VEL
LIN {X 0,Y 312.711,Z 269.153,A -85,B 0,C 180,E1 -15485.159,E2 -15485.159} C_VEL
LIN {X 0,Y 312.849,Z 269.138,A -85,B 0,C 180,E1 -15487.748,E2 -15487.748} C_VEL
LIN {X 0,Y 312.665,Z 269.157,A -85,B 0,C 180,E1 -15491.673,E2 -15491.673} C_VEL
LIN {X 0,Y 312.697,Z 269.156,A -85,B 0,C 180,E1 -15494.889,E2 -15494.889} C_VEL
LIN {X 0,Y 312.606,Z 269.166,A -85,B 0,C 180,E1 -15499.227,E2 -15499.227} C_VEL
LIN {X 0,Y 312.524,Z 269.177,A -85,B 0,C 180,E1 -15502.782,E2 -15502.782} C_VEL
LIN {X 0,Y 312.601,Z 269.173,A -85,B 0,C 180,E1 -15505.937,E2 -15505.937} C_VEL
LIN {X 0,Y 312.546,Z 269.178,A -85,B 0,C 180,E1 -15509.651,E2 -15509.651} C_VEL
LIN {X 0,Y 312.52,Z 269.183,A -85,B 0,C 180,E1 -15513.691,E2 -15513.691} C_VEL
LIN {X 0,Y 312.537,Z 269.179,A -85,B 0,C 180,E1 -15517.385,E2 -15517.385} C_VEL
LIN {X 0,Y 312.491,Z 269.182,A -85,B 0,C 180,E1 -15520.711,E2 -15520.711} C_VEL
LIN {X 0,Y 312.452,Z 269.188,A -85,B 0,C 180,E1 -15524.211,E2 -15524.211} C_VEL
LIN {X 0,Y 312.486,Z 269.187,A -85,B 0,C 180,E1 -15527.92,E2 -15527.92} C_VEL
LIN {X 0,Y 312.508,Z 269.183,A -85,B 0,C 180,E1 -15531.919,E2 -15531.919} C_VEL
LIN {X 0,Y 312.566,Z 269.344,A -85,B 0,C 180,E1 -15535.114,E2 -15535.114} C_VEL
LIN {X 0,Y 315.327,Z 281.351,A -85,B 0,C 180,E1 -15538.507,E2 -15538.507} C_VEL
LIN {X 0,Y 316.953,Z 288.93,A -85,B 0,C 180,E1 -15540.542,E2 -15540.542} C_VEL
LIN {X 0,Y 321.482,Z 301.28,A -85,B 0,C 180,E1 -15541.217,E2 -15541.217} C_VEL
LIN {X 0,Y 326.601,Z 334.299,A -85,B 0,C 180,E1 -15542.407,E2 -15542.407} C_VEL
LIN {X 0,Y 324.237,Z 426.326,A -85,B 0,C 180,E1 -15544.439,E2 -15544.439} C_VEL
LIN {X 0,Y 323.446,Z 440.533,A -85,B 0,C 180,E1 -15544.975,E2 -15544.975} C_VEL
LIN {X 0,Y 322.151,Z 454.858,A -85,B 0,C 180,E1 -15545.77,E2 -15545.77} C_VEL
LIN {X 0,Y 320.776,Z 468.116,A -85,B 0,C 180,E1 -15546.774,E2 -15546.774} C_VEL
LIN {X 0,Y 319.267,Z 480.93,A -85,B 0,C 180,E1 -15548.024,E2 -15548.024} C_VEL
LIN {X 0,Y 317.783,Z 491.383,A -85,B 0,C 180,E1 -15549.277,E2 -15549.277} C_VEL
LIN {X 0,Y 316.223,Z 502.261,A -85,B 0,C 180,E1 -15550.864,E2 -15550.864} C_VEL
LIN {X 0,Y 314.583,Z 513.011,A -85,B 0,C 180,E1 -15552.782,E2 -15552.782} C_VEL
LIN {X 0,Y 313.223,Z 522.737,A -85,B 0,C 180,E1 -15554.923,E2 -15554.923} C_VEL
LIN {X 0,Y 312.304,Z 530.362,A -85,B 0,C 180,E1 -15556.995,E2 -15556.995} C_VEL
LIN {X 0,Y 311.514,Z 536.242,A -85,B 0,C 180,E1 -15558.944,E2 -15558.944} C_VEL
LIN {X 0,Y 311.095,Z 541.084,A -85,B 0,C 180,E1 -15560.901,E2 -15560.901} C_VEL
LIN {X 0,Y 310.819,Z 546.074,A -85,B 0,C 180,E1 -15563.508,E2 -15563.508} C_VEL
LIN {X 0,Y 310.701,Z 549.531,A -85,B 0,C 180,E1 -15566.109,E2 -15566.109} C_VEL
LIN {X 0,Y 310.662,Z 551.567,A -85,B 0,C 180,E1 -15568.704,E2 -15568.704} C_VEL
LIN {X 0,Y 310.693,Z 552.073,A -85,B 0,C 180,E1 -15570,E2 -15570} C_VEL
LIN {X 0,Y 310.673,Z 552.072,A -85,B 0,C 180,E1 -15572.593,E2 -15572.593} C_VEL
LIN {X 0,Y 310.695,Z 550.734,A -85,B 0,C 180,E1 -15575.191,E2 -15575.191} C_VEL
LIN {X 0,Y 310.974,Z 548.047,A -85,B 0,C 180,E1 -15577.793,E2 -15577.793} C_VEL
LIN {X 0,Y 311.541,Z 543.946,A -85,B 0,C 180,E1 -15580.397,E2 -15580.397} C_VEL
LIN {X 0,Y 312.647,Z 538.318,A -85,B 0,C 180,E1 -15582.99,E2 -15582.99} C_VEL
LIN {X 0,Y 313.928,Z 532.004,A -85,B 0,C 180,E1 -15585.251,E2 -15585.251} C_VEL
LIN {X 0,Y 315.657,Z 524.181,A -85,B 0,C 180,E1 -15587.491,E2 -15587.491} C_VEL
LIN {X 0,Y 317.558,Z 516.037,A -85,B 0,C 180,E1 -15589.388,E2 -15589.388} C_VEL
LIN {X 0,Y 319.826,Z 506.256,A -85,B 0,C 180,E1 -15591.258,E2 -15591.258} C_VEL
LIN {X 0,Y 322.189,Z 495.423,A -85,B 0,C 180,E1 -15592.948,E2 -15592.948} C_VEL
LIN {X 0,Y 324.542,Z 483.206,A -85,B 0,C 180,E1 -15594.498,E2 -15594.498} C_VEL
LIN {X 0,Y 326.881,Z 469.995,A -85,B 0,C 180,E1 -15595.809,E2 -15595.809} C_VEL
LIN {X 0,Y 328.839,Z 456.598,A -85,B 0,C 180,E1 -15596.838,E2 -15596.838} C_VEL
LIN {X 0,Y 330.528,Z 442.612,A -85,B 0,C 180,E1 -15597.632,E2 -15597.632} C_VEL
LIN {X 0,Y 331.831,Z 427.869,A -85,B 0,C 180,E1 -15598.2,E2 -15598.2} C_VEL
LIN {X 0,Y 333.003,Z 397.159,A -85,B 0,C 180,E1 -15598.909,E2 -15598.909} C_VEL
LIN {X 0,Y 334.989,Z 336.069,A -85,B 0,C 180,E1 -15600.249,E2 -15600.249} C_VEL
LIN {X 0,Y 330.99,Z 315.087,A -85,B 0,C 180,E1 -15601.278,E2 -15601.278} C_VEL
LIN {X 0,Y 323.638,Z 299.509,A -85,B 0,C 180,E1 -15602.646,E2 -15602.646} C_VEL
LIN {X 0,Y 319.355,Z 291.408,A -85,B 0,C 180,E1 -15603.459,E2 -15603.459} C_VEL
LIN {X 0,Y 317.669,Z 287.867,A -85,B 0,C 180,E1 -15603.822,E2 -15603.822} C_VEL
LIN {X 0,Y 315.434,Z 279.294,A -85,B 0,C 180,E1 -15606.667,E2 -15606.667} C_VEL
LIN {X 0,Y 312.962,Z 270.864,A -85,B 0,C 180,E1 -15609.691,E2 -15609.691} C_VEL
LIN {X 0,Y 312.513,Z 269.174,A -85,B 0,C 180,E1 -15610.362,E2 -15610.362} C_VEL
LIN {X 0,Y 312.535,Z 269.179,A -85,B 0,C 180,E1 -15613.978,E2 -15613.978} C_VEL
LIN {X 0,Y 312.486,Z 269.182,A -85,B 0,C 180,E1 -15617.917,E2 -15617.917} C_VEL
LIN {X 0,Y 312.533,Z 269.179,A -85,B 0,C 180,E1 -15621.909,E2 -15621.909} C_VEL
LIN {X 0,Y 312.504,Z 269.168,A -85,B 0,C 180,E1 -15625.788,E2 -15625.788} C_VEL
LIN {X 0,Y 312.521,Z 269.172,A -85,B 0,C 180,E1 -15628.852,E2 -15628.852} C_VEL
LIN {X 0,Y 312.572,Z 269.169,A -85,B 0,C 180,E1 -15631.823,E2 -15631.823} C_VEL
LIN {X 0,Y 312.582,Z 269.172,A -85,B 0,C 180,E1 -15634.709,E2 -15634.709} C_VEL
LIN {X 0,Y 312.584,Z 269.172,A -85,B 0,C 180,E1 -15637.527,E2 -15637.527} C_VEL
LIN {X 0,Y 312.634,Z 269.168,A -85,B 0,C 180,E1 -15641.655,E2 -15641.655} C_VEL
LIN {X 0,Y 312.689,Z 269.16,A -85,B 0,C 180,E1 -15645.684,E2 -15645.684} C_VEL
LIN {X 0,Y 312.695,Z 269.157,A -85,B 0,C 180,E1 -15649.64,E2 -15649.64} C_VEL
LIN {X 0,Y 312.86,Z 269.128,A -85,B 0,C 180,E1 -15652.252,E2 -15652.252} C_VEL
LIN {X 0,Y 312.71,Z 269.158,A -85,B 0,C 180,E1 -15654.841,E2 -15654.841} C_VEL
LIN {X 0,Y 312.985,Z 269.122,A -85,B 0,C 180,E1 -15658.712,E2 -15658.712} C_VEL
LIN {X 0,Y 313.113,Z 269.104,A -85,B 0,C 180,E1 -15659.998,E2 -15659.998} C_VEL
LIN {X 0,Y 312.93,Z 269.126,A -85,B 0,C 180,E1 -15662.573,E2 -15662.573} C_VEL
LIN {X 0,Y 312.879,Z 269.129,A -85,B 0,C 180,E1 -15666.641,E2 -15666.641} C_VEL
LIN {X 0,Y 312.779,Z 269.142,A -85,B 0,C 180,E1 -15669.048,E2 -15669.048} C_VEL
LIN {X 0,Y 312.624,Z 269.162,A -85,B 0,C 180,E1 -15672.99,E2 -15672.99} C_VEL
LIN {X 0,Y 312.628,Z 269.167,A -85,B 0,C 180,E1 -15675.648,E2 -15675.648} C_VEL
LIN {X 0,Y 312.597,Z 269.17,A -85,B 0,C 180,E1 -15679.707,E2 -15679.707} C_VEL
LIN {X 0,Y 312.537,Z 269.179,A -85,B 0,C 180,E1 -15682.789,E2 -15682.789} C_VEL
LIN {X 0,Y 312.593,Z 269.173,A -85,B 0,C 180,E1 -15685.935,E2 -15685.935} C_VEL
LIN {X 0,Y 312.534,Z 269.167,A -85,B 0,C 180,E1 -15689.649,E2 -15689.649} C_VEL
LIN {X 0,Y 312.507,Z 269.18,A -85,B 0,C 180,E1 -15693.688,E2 -15693.688} C_VEL
LIN {X 0,Y 312.54,Z 269.182,A -85,B 0,C 180,E1 -15697.38,E2 -15697.38} C_VEL
LIN {X 0,Y 312.563,Z 269.37,A -85,B 0,C 180,E1 -15699.731,E2 -15699.731} C_VEL
LIN {X 0,Y 314.106,Z 274.637,A -85,B 0,C 180,E1 -15701.729,E2 -15701.729} C_VEL
LIN {X 0,Y 323.596,Z 291.272,A -85,B 0,C 180,E1 -15703.55,E2 -15703.55} C_VEL
LIN {X 0,Y 331.094,Z 306.267,A -85,B 0,C 180,E1 -15704.931,E2 -15704.931} C_VEL
LIN {X 0,Y 335.69,Z 316.472,A -85,B 0,C 180,E1 -15705.758,E2 -15705.758} C_VEL
LIN {X 0,Y 332.349,Z 410.7,A -85,B 0,C 180,E1 -15707.832,E2 -15707.832} C_VEL
LIN {X 0,Y 331.271,Z 425.087,A -85,B 0,C 180,E1 -15708.38,E2 -15708.38} C_VEL
LIN {X 0,Y 329.758,Z 438.997,A -85,B 0,C 180,E1 -15709.155,E2 -15709.155} C_VEL
LIN {X 0,Y 328.098,Z 451.903,A -85,B 0,C 180,E1 -15710.135,E2 -15710.135} C_VEL
LIN {X 0,Y 326.128,Z 464.214,A -85,B 0,C 180,E1 -15711.323,E2 -15711.323} C_VEL
LIN {X 0,Y 323.81,Z 476.273,A -85,B 0,C 180,E1 -15712.772,E2 -15712.772} C_VEL
LIN {X 0,Y 321.56,Z 487.26,A -85,B 0,C 180,E1 -15714.416,E2 -15714.416} C_VEL
LIN {X 0,Y 319.299,Z 497.215,A -85,B 0,C 180,E1 -15716.237,E2 -15716.237} C_VEL
LIN {X 0,Y 317.236,Z 506.16,A -85,B 0,C 180,E1 -15718.255,E2 -15718.255} C_VEL
LIN {X 0,Y 315.463,Z 513.619,A -85,B 0,C 180,E1 -15720.321,E2 -15720.321} C_VEL
LIN {X 0,Y 313.817,Z 520.41,A -85,B 0,C 180,E1 -15722.672,E2 -15722.672} C_VEL
LIN {X 0,Y 312.718,Z 525.127,A -85,B 0,C 180,E1 -15724.723,E2 -15724.723} C_VEL
LIN {X 0,Y 311.871,Z 528.793,A -85,B 0,C 180,E1 -15726.775,E2 -15726.775} C_VEL
LIN {X 0,Y 311.25,Z 531.558,A -85,B 0,C 180,E1 -15728.822,E2 -15728.822} C_VEL
LIN {X 0,Y 310.761,Z 533.9,A -85,B 0,C 180,E1 -15731.542,E2 -15731.542} C_VEL
LIN {X 0,Y 310.486,Z 534.805,A -85,B 0,C 180,E1 -15734.239,E2 -15734.239} C_VEL
LIN {X 0,Y 310.548,Z 534.308,A -85,B 0,C 180,E1 -15736.921,E2 -15736.921} C_VEL
LIN {X 0,Y 310.559,Z 532.442,A -85,B 0,C 180,E1 -15739.57,E2 -15739.57} C_VEL
LIN {X 0,Y 310.915,Z 529.146,A -85,B 0,C 180,E1 -15742.206,E2 -15742.206} C_VEL
LIN {X 0,Y 311.222,Z 526.225,A -85,B 0,C 180,E1 -15743.886,E2 -15743.886} C_VEL
LIN {X 0,Y 311.691,Z 521.345,A -85,B 0,C 180,E1 -15746.122,E2 -15746.122} C_VEL
LIN {X 0,Y 312.488,Z 515.037,A -85,B 0,C 180,E1 -15748.389,E2 -15748.389} C_VEL
LIN {X 0,Y 313.636,Z 507.189,A -85,B 0,C 180,E1 -15750.642,E2 -15750.642} C_VEL
LIN {X 0,Y 314.907,Z 498.993,A -85,B 0,C 180,E1 -15752.558,E2 -15752.558} C_VEL
LIN {X 0,Y 316.408,Z 489.131,A -85,B 0,C 180,E1 -15754.459,E2 -15754.459} C_VEL
LIN {X 0,Y 317.932,Z 479.02,A -85,B 0,C 180,E1 -15756.059,E2 -15756.059} C_VEL
LIN {X 0,Y 319.522,Z 467.304,A -85,B 0,C 180,E1 -15757.584,E2 -15757.584} C_VEL
LIN {X 0,Y 320.874,Z 455.593,A -85,B 0,C 180,E1 -15758.819,E2 -15758.819} C_VEL
LIN {X 0,Y 322.257,Z 442.775,A -85,B 0,C 180,E1 -15759.889,E2 -15759.889} C_VEL
LIN {X 0,Y 323.325,Z 429.702,A -85,B 0,C 180,E1 -15760.726,E2 -15760.726} C_VEL
LIN {X 0,Y 324.132,Z 415.604,A -85,B 0,C 180,E1 -15761.372,E2 -15761.372} C_VEL
LIN {X 0,Y 324.743,Z 399.09,A -85,B 0,C 180,E1 -15761.825,E2 -15761.825} C_VEL
LIN {X 0,Y 327.091,Z 309.537,A -85,B 0,C 180,E1 -15763.773,E2 -15763.773} C_VEL
LIN {X 0,Y 326.013,Z 305.323,A -85,B 0,C 180,E1 -15763.957,E2 -15763.957} C_VEL
LIN {X 0,Y 317.927,Z 283.9,A -85,B 0,C 180,E1 -15765.13,E2 -15765.13} C_VEL
LIN {X 0,Y 313.592,Z 273.46,A -85,B 0,C 180,E1 -15765.784,E2 -15765.784} C_VEL
LIN {X 0,Y 312.618,Z 269.172,A -85,B 0,C 180,E1 -15767.161,E2 -15767.161} C_VEL
LIN {X 0,Y 312.594,Z 269.173,A -85,B 0,C 180,E1 -15769.709,E2 -15769.709} C_VEL
LIN {X 0,Y 312.522,Z 269.181,A -85,B 0,C 180,E1 -15773.652,E2 -15773.652} C_VEL
LIN {X 0,Y 312.542,Z 269.175,A -85,B 0,C 180,E1 -15776.726,E2 -15776.726} C_VEL
LIN {X 0,Y 312.526,Z 269.176,A -85,B 0,C 180,E1 -15779.235,E2 -15779.235} C_VEL
LIN {X 0,Y 311.854,Z 269.262,A -85,B 0,C 180,E1 -15780.309,E2 -15780.309} C_VEL
LIN {X 0,Y 308.97,Z 269.622,A -85,B 0,C 180,E1 -15782.057,E2 -15782.057} C_VEL
LIN {X 0,Y 306.538,Z 269.927,A -85,B 0,C 180,E1 -15783.474,E2 -15783.474} C_VEL
LIN {X 0,Y 305.516,Z 270.052,A -85,B 0,C 180,E1 -15784.573,E2 -15784.573} C_VEL
LIN {X 0,Y 305.444,Z 270.061,A -85,B 0,C 180,E1 -15784.945,E2 -15784.945} C_VEL
LIN {X 0,Y 305.482,Z 270.055,A -85,B 0,C 180,E1 -15788.54,E2 -15788.54} C_VEL
LIN {X 0,Y 305.51,Z 270.051,A -85,B 0,C 180,E1 -15792.6,E2 -15792.6} C_VEL
LIN {X 0,Y 305.522,Z 270.045,A -85,B 0,C 180,E1 -15796.365,E2 -15796.365} C_VEL
LIN {X 0,Y 305.474,Z 270.056,A -85,B 0,C 180,E1 -15799.898,E2 -15799.898} C_VEL
LIN {X 0,Y 305.489,Z 270.047,A -85,B 0,C 180,E1 -15803.628,E2 -15803.628} C_VEL
LIN {X 0,Y 305.454,Z 270.056,A -85,B 0,C 180,E1 -15806.485,E2 -15806.485} C_VEL
LIN {X 0,Y 305.486,Z 270.055,A -85,B 0,C 180,E1 -15810.952,E2 -15810.952} C_VEL
LIN {X 0,Y 305.562,Z 270.038,A -85,B 0,C 180,E1 -15814.089,E2 -15814.089} C_VEL
LIN {X 0,Y 305.492,Z 270.056,A -85,B 0,C 180,E1 -15818.404,E2 -15818.404} C_VEL
LIN {X 0,Y 305.581,Z 270.044,A -85,B 0,C 180,E1 -15821.219,E2 -15821.219} C_VEL
LIN {X 0,Y 305.641,Z 270.034,A -85,B 0,C 180,E1 -15825.351,E2 -15825.351} C_VEL
LIN {X 0,Y 305.628,Z 270.036,A -85,B 0,C 180,E1 -15829.401,E2 -15829.401} C_VEL
LIN {X 0,Y 305.79,Z 270.012,A -85,B 0,C 180,E1 -15832.076,E2 -15832.076} C_VEL
LIN {X 0,Y 305.681,Z 270.029,A -85,B 0,C 180,E1 -15834.725,E2 -15834.725} C_VEL
LIN {X 0,Y 305.951,Z 270,A -85,B 0,C 180,E1 -15838.686,E2 -15838.686} C_VEL
LIN {X 0,Y 305.951,Z 269.992,A -85,B 0,C 180,E1 -15841.318,E2 -15841.318} C_VEL
LIN {X 0,Y 305.682,Z 270.028,A -85,B 0,C 180,E1 -15845.278,E2 -15845.278} C_VEL
LIN {X 0,Y 305.792,Z 270.018,A -85,B 0,C 180,E1 -15847.928,E2 -15847.928} C_VEL
LIN {X 0,Y 305.599,Z 270.038,A -85,B 0,C 180,E1 -15851.947,E2 -15851.947} C_VEL
LIN {X 0,Y 305.635,Z 270.035,A -85,B 0,C 180,E1 -15855.036,E2 -15855.036} C_VEL
LIN {X 0,Y 305.577,Z 270.042,A -85,B 0,C 180,E1 -15858.785,E2 -15858.785} C_VEL
LIN {X 0,Y 305.484,Z 270.054,A -85,B 0,C 180,E1 -15863.041,E2 -15863.041} C_VEL
LIN {X 0,Y 305.546,Z 270.05,A -85,B 0,C 180,E1 -15866.229,E2 -15866.229} C_VEL
LIN {X 0,Y 305.495,Z 270.054,A -85,B 0,C 180,E1 -15869.052,E2 -15869.052} C_VEL
LIN {X 0,Y 305.448,Z 270.064,A -85,B 0,C 180,E1 -15871.953,E2 -15871.953} C_VEL
LIN {X 0,Y 305.462,Z 270.058,A -85,B 0,C 180,E1 -15875.115,E2 -15875.115} C_VEL
LIN {X 0,Y 305.467,Z 270.058,A -85,B 0,C 180,E1 -15878.534,E2 -15878.534} C_VEL
LIN {X 0,Y 305.456,Z 270.058,A -85,B 0,C 180,E1 -15882.587,E2 -15882.587} C_VEL
LIN {X 0,Y 305.427,Z 270.064,A -85,B 0,C 180,E1 -15886.346,E2 -15886.346} C_VEL
LIN {X 0,Y 305.46,Z 270.062,A -85,B 0,C 180,E1 -15889.894,E2 -15889.894} C_VEL
LIN {X 0,Y 305.511,Z 270.055,A -85,B 0,C 180,E1 -15894.084,E2 -15894.084} C_VEL
LIN {X 0,Y 305.535,Z 270.244,A -85,B 0,C 180,E1 -15894.645,E2 -15894.645} C_VEL
LIN {X 0,Y 308.075,Z 281.381,A -85,B 0,C 180,E1 -15897.879,E2 -15897.879} C_VEL
LIN {X 0,Y 309.644,Z 288.558,A -85,B 0,C 180,E1 -15899.885,E2 -15899.885} C_VEL
LIN {X 0,Y 315.169,Z 303.218,A -85,B 0,C 180,E1 -15900.747,E2 -15900.747} C_VEL
LIN {X 0,Y 320.059,Z 335.525,A -85,B 0,C 180,E1 -15901.935,E2 -15901.935} C_VEL
LIN {X 0,Y 317.671,Z 425.564,A -85,B 0,C 180,E1 -15903.96,E2 -15903.96} C_VEL
LIN {X 0,Y 316.86,Z 440.039,A -85,B 0,C 180,E1 -15904.505,E2 -15904.505} C_VEL
LIN {X 0,Y 315.528,Z 454.442,A -85,B 0,C 180,E1 -15905.315,E2 -15905.315} C_VEL
LIN {X 0,Y 314.056,Z 467.978,A -85,B 0,C 180,E1 -15906.357,E2 -15906.357} C_VEL
LIN {X 0,Y 312.437,Z 481.315,A -85,B 0,C 180,E1 -15907.692,E2 -15907.692} C_VEL
LIN {X 0,Y 310.91,Z 491.665,A -85,B 0,C 180,E1 -15908.971,E2 -15908.971} C_VEL
LIN {X 0,Y 309.418,Z 501.469,A -85,B 0,C 180,E1 -15910.426,E2 -15910.426} C_VEL
LIN {X 0,Y 307.742,Z 512.32,A -85,B 0,C 180,E1 -15912.387,E2 -15912.387} C_VEL
LIN {X 0,Y 306.365,Z 521.7,A -85,B 0,C 180,E1 -15914.471,E2 -15914.471} C_VEL
LIN {X 0,Y 305.407,Z 528.69,A -85,B 0,C 180,E1 -15916.357,E2 -15916.357} C_VEL
LIN {X 0,Y 304.496,Z 535.773,A -85,B 0,C 180,E1 -15918.686,E2 -15918.686} C_VEL
LIN {X 0,Y 304.033,Z 540.673,A -85,B 0,C 180,E1 -15920.688,E2 -15920.688} C_VEL
LIN {X 0,Y 303.731,Z 545.718,A -85,B 0,C 180,E1 -15923.356,E2 -15923.356} C_VEL
LIN {X 0,Y 303.614,Z 549.226,A -85,B 0,C 180,E1 -15926.018,E2 -15926.018} C_VEL
LIN {X 0,Y 303.579,Z 551.309,A -85,B 0,C 180,E1 -15928.673,E2 -15928.673} C_VEL
LIN {X 0,Y 303.605,Z 551.839,A -85,B 0,C 180,E1 -15930,E2 -15930} C_VEL
LIN {X 0,Y 303.597,Z 551.888,A -85,B 0,C 180,E1 -15932.653,E2 -15932.653} C_VEL
LIN {X 0,Y 303.622,Z 550.607,A -85,B 0,C 180,E1 -15935.312,E2 -15935.312} C_VEL
LIN {X 0,Y 303.915,Z 547.977,A -85,B 0,C 180,E1 -15937.975,E2 -15937.975} C_VEL
LIN {X 0,Y 304.528,Z 543.928,A -85,B 0,C 180,E1 -15940.639,E2 -15940.639} C_VEL
LIN {X 0,Y 305.321,Z 539.911,A -85,B 0,C 180,E1 -15942.631,E2 -15942.631} C_VEL
LIN {X 0,Y 306.457,Z 534.947,A -85,B 0,C 180,E1 -15944.611,E2 -15944.611} C_VEL
LIN {X 0,Y 308.03,Z 527.862,A -85,B 0,C 180,E1 -15946.913,E2 -15946.913} C_VEL
LIN {X 0,Y 310.16,Z 519.142,A -85,B 0,C 180,E1 -15949.181,E2 -15949.181} C_VEL
LIN {X 0,Y 312.384,Z 510.047,A -85,B 0,C 180,E1 -15951.097,E2 -15951.097} C_VEL
LIN {X 0,Y 314.988,Z 499.056,A -85,B 0,C 180,E1 -15952.982,E2 -15952.982} C_VEL
LIN {X 0,Y 317.385,Z 488,A -85,B 0,C 180,E1 -15954.515,E2 -15954.515} C_VEL
LIN {X 0,Y 319.383,Z 477.413,A -85,B 0,C 180,E1 -15955.724,E2 -15955.724} C_VEL
LIN {X 0,Y 321.424,Z 465.64,A -85,B 0,C 180,E1 -15956.805,E2 -15956.805} C_VEL
LIN {X 0,Y 323.424,Z 452.176,A -85,B 0,C 180,E1 -15957.764,E2 -15957.764} C_VEL
LIN {X 0,Y 325.008,Z 438.083,A -85,B 0,C 180,E1 -15958.494,E2 -15958.494} C_VEL
LIN {X 0,Y 326.036,Z 424.576,A -85,B 0,C 180,E1 -15958.968,E2 -15958.968} C_VEL
LIN {X 0,Y 329.1,Z 337.13,A -85,B 0,C 180,E1 -15960.929,E2 -15960.929} C_VEL
LIN {X 0,Y 325.428,Z 317.821,A -85,B 0,C 180,E1 -15961.909,E2 -15961.909} C_VEL
LIN {X 0,Y 317.192,Z 300.537,A -85,B 0,C 180,E1 -15963.504,E2 -15963.504} C_VEL
LIN {X 0,Y 311.848,Z 290.652,A -85,B 0,C 180,E1 -15964.569,E2 -15964.569} C_VEL
LIN {X 0,Y 310.392,Z 287.555,A -85,B 0,C 180,E1 -15964.917,E2 -15964.917} C_VEL
LIN {X 0,Y 307.721,Z 277.577,A -85,B 0,C 180,E1 -15968.417,E2 -15968.417} C_VEL
LIN {X 0,Y 305.497,Z 270.047,A -85,B 0,C 180,E1 -15971.334,E2 -15971.334} C_VEL
LIN {X 0,Y 305.463,Z 270.063,A -85,B 0,C 180,E1 -15974.499,E2 -15974.499} C_VEL
LIN {X 0,Y 305.442,Z 270.06,A -85,B 0,C 180,E1 -15978.142,E2 -15978.142} C_VEL
LIN {X 0,Y 305.493,Z 270.058,A -85,B 0,C 180,E1 -15981.599,E2 -15981.599} C_VEL
LIN {X 0,Y 305.46,Z 270.034,A -85,B 0,C 180,E1 -15984.885,E2 -15984.885} C_VEL
LIN {X 0,Y 305.45,Z 270.055,A -85,B 0,C 180,E1 -15988.353,E2 -15988.353} C_VEL
LIN {X 0,Y 305.518,Z 270.053,A -85,B 0,C 180,E1 -15991.112,E2 -15991.112} C_VEL
LIN {X 0,Y 305.569,Z 270.049,A -85,B 0,C 180,E1 -15994.086,E2 -15994.086} C_VEL
LIN {X 0,Y 305.496,Z 270.055,A -85,B 0,C 180,E1 -15998.401,E2 -15998.401} C_VEL
LIN {X 0,Y 305.586,Z 270.042,A -85,B 0,C 180,E1 -16001.216,E2 -16001.216} C_VEL
LIN {X 0,Y 305.644,Z 270.034,A -85,B 0,C 180,E1 -16005.347,E2 -16005.347} C_VEL
LIN {X 0,Y 305.632,Z 270.033,A -85,B 0,C 180,E1 -16009.398,E2 -16009.398} C_VEL
LIN {X 0,Y 305.802,Z 270.008,A -85,B 0,C 180,E1 -16012.072,E2 -16012.072} C_VEL
LIN {X 0,Y 305.681,Z 270.033,A -85,B 0,C 180,E1 -16014.722,E2 -16014.722} C_VEL
LIN {X 0,Y 305.952,Z 269.998,A -85,B 0,C 180,E1 -16018.682,E2 -16018.682} C_VEL
LIN {X 0,Y 305.951,Z 269.989,A -85,B 0,C 180,E1 -16021.314,E2 -16021.314} C_VEL
LIN {X 0,Y 305.838,Z 270.007,A -85,B 0,C 180,E1 -16026.596,E2 -16026.596} C_VEL
LIN {X 0,Y 305.727,Z 270.019,A -85,B 0,C 180,E1 -16029.258,E2 -16029.258} C_VEL
LIN {X 0,Y 305.579,Z 270.037,A -85,B 0,C 180,E1 -16033.294,E2 -16033.294} C_VEL
LIN {X 0,Y 305.584,Z 270.045,A -85,B 0,C 180,E1 -16036.019,E2 -16036.019} C_VEL
LIN {X 0,Y 305.571,Z 270.046,A -85,B 0,C 180,E1 -16039.446,E2 -16039.446} C_VEL
LIN {X 0,Y 305.482,Z 270.055,A -85,B 0,C 180,E1 -16043.041,E2 -16043.041} C_VEL
LIN {X 0,Y 305.537,Z 270.049,A -85,B 0,C 180,E1 -16046.226,E2 -16046.226} C_VEL
LIN {X 0,Y 305.485,Z 270.053,A -85,B 0,C 180,E1 -16049.049,E2 -16049.049} C_VEL
LIN {X 0,Y 305.453,Z 270.061,A -85,B 0,C 180,E1 -16053.516,E2 -16053.516} C_VEL
LIN {X 0,Y 305.49,Z 270.054,A -85,B 0,C 180,E1 -16056.734,E2 -16056.734} C_VEL
LIN {X 0,Y 305.494,Z 270.225,A -85,B 0,C 180,E1 -16058.764,E2 -16058.764} C_VEL
LIN {X 0,Y 306.917,Z 274.909,A -85,B 0,C 180,E1 -16060.627,E2 -16060.627} C_VEL
LIN {X 0,Y 309.279,Z 278.878,A -85,B 0,C 180,E1 -16061.119,E2 -16061.119} C_VEL
